(****************************************************************************************)
(* POU:		HLI3_HandlePlcSpindle                      									*)
(* Type:	Function Block																*)
(* Author: 	HR, MiB, TV																    *)
(* Date: 	10/11/10																	*)
(* Rev.: 	1.0																			*)
(* Rev.: 	1.6	14/10/23    															*)
(* ------------------------------------------------------------------------------------ *)
(* Desc:	Function block for handling technology functions of PLC spindles. It works	*)
(*			properly if there is a ation axis in the configuration. The logical 		*)
(*			axis no. 'n' of that axis is used to indetify that spindle in this function	*)
(*			block. This implies a spindle configuration like the folowing:				*)
(*				spdl_anzahl                         1	(maybe more?)					*)
(*				main_spindle_ax_nr                  n	(enter right value there)		*)
(*				main_spindle_name                   S									*)
(*				spindle_m_fct_free                  0									*)
(*				spindel[0].bezeichnung              S1									*)
(*				spindel[0].log_achs_nr              n	(enter right value there)		*)
(*				spindel[0].plc_control              1									*)
(*																						*)
(*			The function block may raise some errors specified by an error id:			*)
(*				+ 10000: axis number not valid!											*)
(*																						*)
(****************************************************************************************)
(* Date:	13/09/16																	*)
(* Author:	RCH																			*)
(* Rev:		1.1																			*)
(* ------------------------------------------------------------------------------------ *)
(* Desc 	Renamed, according to Tc2 version. This FB also works for CNC spindles with	*) 
(*			S or M functions set to inform PLC. 										*)
(****************************************************************************************)
(* Date:	13/09/16																	*)
(* Author:	RCH																			*)
(* Rev:		1.2																			*)
(* ------------------------------------------------------------------------------------ *)
(* Desc 	Introduced new input parameters 'bIsChannelSpecific' and 'nChannelNo' in 	*)
(*			order to make this FB work for PLC spindles which are sending synch.		*)
(*			requests via the channel specific section of the HLI. Here the spindle		*)
(* 			specific parameters have to be set as follows:								*)
(*				spindel[n].plc_control            1			(P-CHAN-00069)				*)
(*				spindel[n].log_achs_nr            m			(P-CHAN-00036)				*)
(*																						*)
(*			The logical axis number in P-CHAN-00036 used for such a spindle must not be	*)
(*			lower than one and must not be used by any other axis. This FB works if the	*)
(*			value of this logical axis number fits the parameter 'nHliAxisIdx' only!	*)
(* 																						*)
(*			In order to guarantee save HLI access the following new error codes have	*)
(*			been introduced:															*)
(*				+ 20000: Channel no lower than one!										*)
(*				+ 20001: Channel number exceeds number of configured channels.			*)
(*				+ 20002: No HLI data for channel.										*)
(****************************************************************************************)
(* Date:	14/01/22																	*)
(* Author:	TV																			*)
(* Rev:		1.3																			*)
(* ------------------------------------------------------------------------------------ *)
(* Desc:	bugfix in function to check nHLIAxisIdx and LogAxisId						*) 
(****************************************************************************************)
(* Date:	14/09/10																	*)
(* Author:	RCH																			*)
(* Rev:		1.4																			*)
(* ------------------------------------------------------------------------------------ *)
(* Desc 	Added optional handling of spindle gear change M functions M40 - M45.		*)
(****************************************************************************************)
(* Date:	14/09/12																	*)
(* Author:	RCH																			*)
(* Rev:		1.5																			*)
(* ------------------------------------------------------------------------------------ *)
(* Desc 	Fixed bug with spindle M functions send by the channel spec. section of the	*)
(*			HLI. So far the channel specific section was used for determining the value *)
(*			of  'nTechFctMaxidx'.														*)
(****************************************************************************************)
(* Date:	14/10/23																	*)
(* Author:	MiB																			*)
(* Rev:		1.6																			*)
(* ------------------------------------------------------------------------------------ *)
(* Desc 	Introduced parameter "nLogAxisNoChannelSpecific" which allows to use a plc  *)
(*			spindle without a simulation axis for the spindle. 				 			*)
(*			This paramater is only used if "bIsChannelSpecific == true"					*)
(*																						*)
(*				spindel[n].plc_control            1			(P-CHAN-00069)				*)
(*				spindel[n].log_achs_nr            m			(P-CHAN-00036)				*)
(*																						*)
(*			The logical axis number in P-CHAN-00036 used for such a spindle must not be	*)
(*			lower than one and must not be used by any other axis. This FB works if the	*)
(*			value of this logical axis number fits the parameter 						*)
(*			'nLogAxisNoChannelSpecific' only!											*)
(****************************************************************************************)
(* Date:	15/03/05																	*)
(* Author:	MiB																			*)
(* Rev:		1.7																			*)
(* ------------------------------------------------------------------------------------ *)
(* Desc 	Removed gearchange m functions from var_in_out							    *)
(*			Created new FB HLI3_SpindleTechnoGearchange									*)
(****************************************************************************************)
(*								Init Pointer to pM40..pM45								*)
(****************************************************************************************)
(* Date:	17/02/03																	*)
(* Author:	MiB																			*)
(* Rev:		1.7																			*)
(* ------------------------------------------------------------------------------------ *)
(* Desc 	Handling of late sync M functions. 											*)
(*			Usage of different structure TECHNO_UNIT_AX and TECHNO_UNIT_CH, depending 	*)
(*			on channel or axis specific specific interface 							 	*)
(****************************************************************************************)
(* Date:	19/04/19																	*)
(* Author:	TV																			*)
(* Rev:		1.8																			*)
(* ------------------------------------------------------------------------------------ *)
(* Desc 	Reset the M-Function flags after Reset										*)
(****************************************************************************************)


IF bFirstRun THEN
	bFirstRun := FALSE;
	pM40 := ADR(dummyM40);
	pM41 := ADR(dummyM41);
	pM42 := ADR(dummyM42);
	pM43 := ADR(dummyM43);
	pM44 := ADR(dummyM44);
	pM45 := ADR(dummyM45);	
END_IF

A_HandleTechno();

ACTION A_HandleTechno:

(****************************************************************************************)
(*								Cyclic reset of  error flag 							*)
(****************************************************************************************)
bError										:= FALSE;
nErrorId									:= 0;

(****************************************************************************************)
(*							  Check for valid logical axis no.							*)
(****************************************************************************************)
IF NOT bIsChannelSpecific AND NOT HLI3_CheckAxisValid(nHliAxisIdx := nHliAxisIdx) THEN
	bError									:= TRUE;
	nErrorId								:= 10000;
	RETURN;
END_IF

IF NOT HLI3_CheckChannelValid(nChannel := nHliChannelIdx) THEN
	bError									:= TRUE;
	nErrorId								:= 20000;
	RETURN;	
END_IF

(****************************************************************************************)
(*											Reset										*)
(****************************************************************************************)
fbRtrigChannelReset
	(CLK := bChannelReset);

IF fbRtrigChannelReset.Q THEN
	M_Reset(M03:=M03, M04:=M04,M05:=M05,M19:=M19);
END_IF

(****************************************************************************************)
(*									Receive requests from cnc							*)
(****************************************************************************************)
(* Look out for open technology function either on the channel or the axis specific		*)
(* section of the HLI, depending on parameter ''.										*)
IF bIsChannelSpecific THEN
	nOpenTechnoCount	:= gpCh[nHliChannelIdx]^.used_units_std_sync_r;
	nOpenTechnoCountLate:= gpCh[nHliChannelIdx]^.used_units_late_sync_r;
	
	nTechFctMaxidx 		:= gpCh[nHliChannelIdx]^.used_units_std_sync_r - 1;
	nTechFctMaxIdxLate 	:= gpCh[nHliChannelIdx]^.used_units_late_sync_r - 1;
ELSE
	nOpenTechnoCount	:= gpAx[nHliAxisIdx]^.used_units_std_sync_r;
	nOpenTechnoCountLate:= gpAx[nHliAxisIdx]^.used_units_late_sync_r;

	nTechFctMaxidx 		:= gpAx[nHliAxisIdx]^.used_units_std_sync_r - 1;
	nTechFctMaxIdxLate 	:= gpAx[nHliAxisIdx]^.used_units_late_sync_r - 1;		
END_IF

IF nOpenTechnoCount > 0 THEN
	FOR nLoop := 0 TO nTechFctMaxIdx DO
		(* Depending on the source determined by parameter 'bIsChannelSpecific', the		*)
		(* channel or axis specific section of the HLI will be examined.					*)
		IF bIsChannelSpecific THEN		
				
			M_HandleTechnoCh(ADR(gpCh[nHliChannelIdx]^.techno_unit_std_sync[nLoop]), M03 := M03, M04 := M04, M05 := M05, M19 := M19);												
		ELSE
			(* Get current axis specifc technology data *)			
			M_HandleTechnoAx(ADR(gpAx[nHliAxisIdx]^.techno_unit_std_sync[nLoop]), M03 := M03, M04 := M04, M05 := M05, M19 := M19);		
		END_IF																	
	END_FOR	
END_IF

IF nOpenTechnoCountLate > 0 THEN
	FOR nLoop := 0 TO nTechFctMaxIdxLate DO
		(* Depending on the source determined by parameter 'bIsChannelSpecific', the		*)
		(* channel or axis specific section of the HLI will be examined.					*)
		IF bIsChannelSpecific THEN			
			M_HandleTechnoCh(ADR(gpCh[nHliChannelIdx]^.techno_unit_late_sync[nLoop]), M03 := M03, M04 := M04, M05 := M05, M19 := M19);						
		ELSE
			(* Get current axis specifc technology data *)			
			M_HandleTechnoAx(ADR(gpAx[nHliAxisIdx]^.techno_unit_late_sync[nLoop]), M03 := M03, M04 := M04, M05 := M05, M19 := M19);	
		END_IF																	
	END_FOR	
END_IF

IF nOpenTechnoCountLate  = 0 AND nOpenTechnoCount = 0 THEN	
	M_Reset(M03:=M03, M04:=M04,M05:=M05,M19:=M19); 	 	
END_IF
END_ACTION

METHOD PROTECTED M_HandleTechnoAx
VAR_INPUT
	pActTechnoUnit:	POINTER TO TECHNO_UNIT_AX;	
END_VAR
VAR_IN_OUT
	/// Raises if the cnc program encounters a M03 for the relevant spindle. Reset this for acknowledge 
	M03: BOOL;
	/// Raises if the cnc program encounters a M04 for the relevant spindle. Reset this for acknowledge 
	M04: BOOL;
	/// Raises if the cnc program encounters a M05 for the relevant spindle. Reset this for acknowledge 
	M05: BOOL;
	/// Raises if the cnc program encounters a M19 for the relevant spindle. Reset this for acknowledge 
	M19: BOOL;
END_VAR
		
		(* Check request *)
		IF pActTechnoUnit^.please_rw AND
		   NOT pActTechnoUnit^.done_w
		THEN
			CASE UINT_TO_UDINT(pActTechnoUnit^.fkt_ctrl_r) OF
		     (* -------------------------------------------------------------------------- *)
			 (* Handle M function *)
			 HLI_INTF_M_FKT:
				pMProcess					:= ADR(pActTechnoUnit^.attribut_r.data[0]);
				
				IF (pMProcess > 0) AND bHandleGearChange THEN
					CASE pMProcess^.nr OF
					 40:	M_ManageAcknowledgement(ADR(M40_Internal), pM40, ADR(bAcknowledge));
					 41:	M_ManageAcknowledgement(ADR(M41_Internal), pM41, ADR(bAcknowledge));
					 42:	M_ManageAcknowledgement(ADR(M42_Internal), pM42, ADR(bAcknowledge));
					 43:	M_ManageAcknowledgement(ADR(M43_Internal), pM43, ADR(bAcknowledge));
					 44:	M_ManageAcknowledgement(ADR(M44_Internal), pM44, ADR(bAcknowledge));
					 45:	M_ManageAcknowledgement(ADR(M45_Internal), pM45, ADR(bAcknowledge));
					END_CASE
				END_IF
				
			 (* -------------------------------------------------------------------------- *)
			 (* Handle S function *)
			 HLI_INTF_SPINDEL:
				pSProcess					:= ADR(pActTechnoUnit^.attribut_r.data[0]);
				
				(* If we are working with spindle functions provided by the channel 		*)
				(* specific section of the HLI the logical axis number transmitted from the *)
				(* CNC must fit the one given in parameter 'nLogAxisNoChannelSpecific'!					*)												
				IF bIsChannelSpecific AND (UINT_TO_INT(pSProcess^.log_achs_nr) <> nLogAxisNoChannelSpecific) THEN
					RETURN;
				END_IF
	
				CASE pSProcess^.move_cmd OF
				 (* ----------------------------------------------------------------------- *)
				 0: (* M19 *)
					IF (pSProcess^.pos_cmd = 19) AND
					   NOT M19_Internal THEN
						nPosition			:= pSProcess^.pos;
						M19_Internal		:= TRUE;
						M19					:= TRUE;
					ELSE
						IF NOT M19 THEN
							M19_Internal	:= FALSE;
							bAcknowledge	:= TRUE;
						END_IF
					END_IF
	
				 (* ----------------------------------------------------------------------- *)
				 3: (* M03 *)
					nRevolution				:= pSProcess^.rev;
	
					IF NOT M03_Internal THEN
						M03_Internal		:= TRUE;
						M03					:= TRUE;
					ELSE
						IF NOT M03 THEN
							M03_Internal	:= FALSE;
							bAcknowledge	:= TRUE;
						END_IF
					END_IF
	
				 (* ----------------------------------------------------------------------- *)
				 4: (* M04 *)
					nRevolution				:= pSProcess^.rev;
	
					IF NOT M04_Internal THEN
						M04_Internal		:= TRUE;
						M04					:= TRUE;
					ELSE
						IF NOT M04 THEN
							M04_Internal	:= FALSE;
							bAcknowledge	:= TRUE;
						END_IF
					END_IF
	
				 (* ----------------------------------------------------------------------- *)
				 5: (* M05 *)
					IF NOT M05_Internal THEN
						M05_Internal		:= TRUE;
						M05					:= TRUE;
					ELSE
						IF NOT M05 THEN
							M05_Internal	:= FALSE;
							bAcknowledge	:= TRUE;
						END_IF
					END_IF
	
				END_CASE
			END_CASE
	
			(* Handle acknowledgement *)
			IF bAcknowledge THEN
				bAcknowledge				:= FALSE;
				nRevolution					:= 0;
				nPosition					:= 0;
				pActTechnoUnit^.please_rw 	:= FALSE;
		   		pActTechnoUnit^.done_w		:= TRUE;
			END_IF
		END_IF
END_METHOD

METHOD PROTECTED M_HandleTechnoCh
VAR_INPUT
	pActTechnoUnit:	POINTER TO TECHNO_UNIT_CH;
END_VAR
VAR_IN_OUT
	/// Raises if the cnc program encounters a M03 for the relevant spindle. Reset this for acknowledge 
	M03: BOOL;
	/// Raises if the cnc program encounters a M04 for the relevant spindle. Reset this for acknowledge 
	M04: BOOL;
	/// Raises if the cnc program encounters a M05 for the relevant spindle. Reset this for acknowledge 
	M05: BOOL;
	/// Raises if the cnc program encounters a M19 for the relevant spindle. Reset this for acknowledge 
	M19: BOOL;
END_VAR
		
		(* Check request *)
		IF pActTechnoUnit^.please_rw AND
		   NOT pActTechnoUnit^.done_w
		THEN
			CASE UINT_TO_UDINT(pActTechnoUnit^.fkt_ctrl_r) OF
		     (* -------------------------------------------------------------------------- *)
			 (* Handle M function *)
			 HLI_INTF_M_FKT:
				pMProcess					:= ADR(pActTechnoUnit^.attribut_r.data[0]);
				
				IF (pMProcess > 0) AND bHandleGearChange THEN
					CASE pMProcess^.nr OF
					 40:	M_ManageAcknowledgement(ADR(M40_Internal), pM40, ADR(bAcknowledge));
					 41:	M_ManageAcknowledgement(ADR(M41_Internal), pM41, ADR(bAcknowledge));
					 42:	M_ManageAcknowledgement(ADR(M42_Internal), pM42, ADR(bAcknowledge));
					 43:	M_ManageAcknowledgement(ADR(M43_Internal), pM43, ADR(bAcknowledge));
					 44:	M_ManageAcknowledgement(ADR(M44_Internal), pM44, ADR(bAcknowledge));
					 45:	M_ManageAcknowledgement(ADR(M45_Internal), pM45, ADR(bAcknowledge));
					END_CASE
				END_IF
				
			 (* -------------------------------------------------------------------------- *)
			 (* Handle S function *)
			 HLI_INTF_SPINDEL:
				pSProcess					:= ADR(pActTechnoUnit^.attribut_r.data[0]);
				
				(* If we are working with spindle functions provided by the channel 		*)
				(* specific section of the HLI the logical axis number transmitted from the *)
				(* CNC must fit the one given in parameter 'nLogAxisNoChannelSpecific'!					*)												
				IF bIsChannelSpecific AND (UINT_TO_INT(pSProcess^.log_achs_nr) <> nLogAxisNoChannelSpecific) THEN
					RETURN;
				END_IF
	
				CASE pSProcess^.move_cmd OF
				 (* ----------------------------------------------------------------------- *)
				 0: (* M19 *)
					IF (pSProcess^.pos_cmd = 19) AND
					   NOT M19_Internal THEN
						nPosition			:= pSProcess^.pos;
						M19_Internal		:= TRUE;
						M19					:= TRUE;
					ELSE
						IF NOT M19 THEN
							M19_Internal	:= FALSE;
							bAcknowledge	:= TRUE;
						END_IF
					END_IF
	
				 (* ----------------------------------------------------------------------- *)
				 3: (* M03 *)
					nRevolution				:= pSProcess^.rev;
	
					IF NOT M03_Internal THEN
						M03_Internal		:= TRUE;
						M03					:= TRUE;
					ELSE
						IF NOT M03 THEN
							M03_Internal	:= FALSE;
							bAcknowledge	:= TRUE;
						END_IF
					END_IF
	
				 (* ----------------------------------------------------------------------- *)
				 4: (* M04 *)
					nRevolution				:= pSProcess^.rev;
	
					IF NOT M04_Internal THEN
						M04_Internal		:= TRUE;
						M04					:= TRUE;
					ELSE
						IF NOT M04 THEN
							M04_Internal	:= FALSE;
							bAcknowledge	:= TRUE;
						END_IF
					END_IF
	
				 (* ----------------------------------------------------------------------- *)
				 5: (* M05 *)
					IF NOT M05_Internal THEN
						M05_Internal		:= TRUE;
						M05					:= TRUE;
					ELSE
						IF NOT M05 THEN
							M05_Internal	:= FALSE;
							bAcknowledge	:= TRUE;
						END_IF
					END_IF
	
				END_CASE
			END_CASE
	
			(* Handle acknowledgement *)
			IF bAcknowledge THEN
				bAcknowledge				:= FALSE;
				nRevolution					:= 0;
				nPosition					:= 0;
				pActTechnoUnit^.please_rw 	:= FALSE;
		   		pActTechnoUnit^.done_w		:= TRUE;
			END_IF
		END_IF
END_METHOD

{attribute 'object_name' := 'M_ManageAcknowledgement'}
METHOD PRIVATE M_ManageAcknowledgement
VAR_INPUT
	pInternal: POINTER TO BOOL;
	pPublic: POINTER TO BOOL;
	pAcknowledgement: POINTER TO BOOL;
END_VAR
IF NOT pInternal^ THEN
	pInternal^			:= TRUE;
	pPublic^			:= TRUE;	
ELSIF NOT pPublic^ THEN
	pInternal^			:= FALSE;
	pAcknowledgement^	:= TRUE;
END_IF
END_METHOD

METHOD M_Reset : BOOL
VAR_INPUT
END_VAR
VAR_IN_OUT	 
	M03: BOOL;	 
	M04: BOOL;	 
	M05: BOOL;	 
	M19: BOOL;
END_VAR
	nRevolution		:= 0;
	nPosition		:= 0;
	bAcknowledge	:= FALSE;
	M03				:= FALSE;
	M03_Internal	:= FALSE;
	M04				:= FALSE;
	M04_Internal	:= FALSE;
	M05				:= FALSE;
	M05_Internal	:= FALSE;
	M19				:= FALSE;
	M19_Internal	:= FALSE;	
	pM40^			:= FALSE;
	M40_Internal	:= FALSE;
	pM41^			:= FALSE;
	M41_Internal	:= FALSE;
	pM42^			:= FALSE;
	M42_Internal	:= FALSE;
	pM43^			:= FALSE;
	M43_Internal	:= FALSE;
	pM44^			:= FALSE;
	M44_Internal	:= FALSE;
	pM45^			:= FALSE;
	M45_Internal	:= FALSE;
END_METHOD

END_FUNCTION_BLOCK

// CNC/13 Spindle/HLI3_HandleSpindleTechnoGearchange
FUNCTION_BLOCK HLI3_HandleSpindleTechnoGearchange EXTENDS HLI3_HandleSpindleTechno
VAR_INPUT
END_VAR
VAR_OUTPUT
END_VAR
VAR_IN_OUT
		/// Raises if the cnc program encounters a M40 for the relevant spindle. Reset this for acknowledge 
	M40: BOOL;
	/// Raises if the cnc program encounters a M41 for the relevant spindle. Reset this for acknowledge 
	M41: BOOL;
	/// Raises if the cnc program encounters a M42 for the relevant spindle. Reset this for acknowledge 
	M42: BOOL;
	/// Raises if the cnc program encounters a M43 for the relevant spindle. Reset this for acknowledge 
	M43: BOOL;
	/// Raises if the cnc program encounters a M44 for the relevant spindle. Reset this for acknowledge 
	M44: BOOL;
	/// Raises if the cnc program encounters a M45 for the relevant spindle. Reset this for acknowledge 
	M45: BOOL;	
END_VAR
VAR
END_VAR

(* Date:	15/03/05																	*)
(* Author:	MiB																			*)
(* Rev:		1.0																			*)
(* ------------------------------------------------------------------------------------ *)
(* Desc 	Handling of spindle gear change M functions M40 - M45.						*)
(*			extends HLI3_SpindleTechno													*)
(*			overwrites the internal pointers to M40..M45 to VAR_IN_OUT					*)


SUPER^.pM40 := ADR(M40);
SUPER^.pM41 := ADR(M41);
SUPER^.pM42 := ADR(M42);
SUPER^.pM43 := ADR(M43);
SUPER^.pM44 := ADR(M44);
SUPER^.pM45 := ADR(M45);

A_HandleTechno();

END_FUNCTION_BLOCK

// CNC/13 Spindle/HLI3_MoveSpindle
///*********************************************************************************************************
///NAME.......................:	HLI3_MoveSpindle	
///DATUM....................:	24.5.2018
///AUTOR....................:	Michael Balsfulland (MiB) / TV
///VERSION................:	1.1
///				1.0 24.05.2018 Kopie von HLI_MoveSpindle
///				1.1 03.03.2019 Parametrierung der ControlUnit erst wenn command_semaphor_rw = false
 ///BESCHREIBUNG.:	 Spindel mit einer vorgegeben Geschwindigkeit starten oder Spindel stoppen
///......................: 	
///
///**********************************************************************************************************
 FUNCTION_BLOCK HLI3_MoveSpindle
VAR_INPUT
	/// HLI Index 
	nHliAxisIdx: INT;
	/// U/min 
	nSpeed: DINT;		// [u/min]
	/// steigende Flanke 
	bStart: BOOL;
	/// steigende Flanke 
	bStop: BOOL;
END_VAR
VAR_OUTPUT
	bBusy: BOOL;
	bError: BOOL;
	nErrID: INT;
	sErrText: STRING;
END_VAR
VAR
	pUnit: POINTER TO MC_CONTROL_EXT_TO_IPO;
	fbRTrigStart: R_TRIG;
	fbRTrigStop: R_TRIG;
	nState: INT;	 	
END_VAR

IF NOT (HLI3_CheckAxisValid(nHliAxisIdx := nHliAxisIdx)) THEN
		nState := -1;
		nErrID := 2;
		sErrText := 'Achsstruktur nicht vorhanden -> eventuell HLI Init nicht OK';
	RETURN;
END_IF

fbRTrigStart(clk := bStart);
IF fbRTrigStart.Q THEN
	bError := FALSE;
	nErrId := 0;
	sErrText := '';
	nState := 100;   (* Spindel starten *)
END_IF


fbRTrigStop(clk := bStop);
IF fbRTrigStop.Q THEN
	bError := FALSE;
	nErrId := 0;
	sErrText := '';
	nState := 200;  (* Spindel stoppen *)
END_IF

IF fbRTrigStop.Q OR fbRTrigStart.Q THEN   (* Grundzustände testen *)
	bBusy := TRUE;		
	IF gpAx[nHliAxisIdx]^.ipo_state.spindle_axis_r <> TRUE THEN
		nState := -1;
		nErrID := 3;
		sErrText := 'Achse ist kene Spindel';
	END_IF
END_IF

CASE nState OF


-1: (* Fehler *)
   	bError := TRUE;
	bBusy := FALSE;

0: (* IDLE *)
	bBusy := FALSE;


100: (* Spindel starten *)
	(* Check Override *)
	gpAx[nHliAxisIdx]^.ipo_mc_control.override.enable_w := TRUE;
	IF gpAx[nHliAxisIdx]^.ipo_mc_control.override.state_r = 0 THEN
		nState := -1;
		nErrID := 4;
		sErrText := 'Spindeloverride = 0';
	ELSE
		nState := 110;
	END_IF


110: (* Parametrieren des Aufrufs *)
	pUnit := ADR(gpAx[nHliAxisIdx]^.ipo_mc_control.ext_to_ipo);
	IF pUnit^.command_semaphor_rw = FALSE THEN
		IF (nSpeed > 0) THEN
			pUnit^.command_w.vb_prog   :=  nSpeed * 360 / 60 * 1000  ;(*Programmierter Satzvorschub in u/min*)
			pUnit^.command_w.dreh_info := 1;(* rechtslauf *)
		ELSE
			pUnit^.command_w.vb_prog   :=  -nSpeed * 360 / 60 * 1000  ;(*Programmierter Satzvorschub in u/min*)
			pUnit^.command_w.dreh_info := 0;(* linkslauf*)
		END_IF
		pUnit^.command_w.geo_gm_fkt    := 0;(*G- und M- Fkt.-Bitleiste*)
		pUnit^.command_w.satz_typ      := HLI_NC_MOVE_ENDLOS;(*Einer der Werte: HLI_NC_MOVE_LIN, HLI_NC_MOVREF, HLI_NC_MOVE_ENDLOS, HLI_NC_SPINDEL_STOP*)
		pUnit^.command_w.job_nr		   := 0;
		pUnit^.command_w.job_ackn      := FALSE;
	    pUnit^.command_semaphor_rw     := TRUE;
	    nState := 120;
	END_IF

	IF (nSpeed=0) THEN
		nState := -1;
		nErrID := 6;
		sErrText := 'Vorgabegeschwindigkeit = 0';
	END_IF

120: (* Start *)

	IF pUnit^.command_semaphor_rw = FALSE THEN
	    nState := 300;  (* checken Auftragsfehler *)
	END_IF



200: (* Spindel Stopp*)
	pUnit := ADR(gpAx[nHliAxisIdx]^.ipo_mc_control.ext_to_ipo);
	IF pUnit^.command_semaphor_rw = FALSE THEN
		pUnit^.command_w.satz_typ  := HLI_NC_SPINDEL_STOP;(*Einer der Werte: HLI_NC_MOVE_LIN, HLI_NC_MOVREF, HLI_NC_MOVE_ENDLOS, HLI_NC_SPINDEL_STOP*)		
		pUnit^.command_w.job_nr		   := 0;
		pUnit^.command_w.job_ackn      := FALSE;
		pUnit^.command_w.dreh_info := 0;(*Drehinformation*)
	   	pUnit^.command_semaphor_rw := TRUE;
	   	nState := 210;
	END_IF

210: (* Warten auf Stop *)
	IF pUnit^.command_semaphor_rw = FALSE THEN
	    nState := 300;   (* checken Auftragsfehler *)
	END_IF

300: (* checken Auftragsfehler *)
	IF (gpAx[nHliAxisIdx]^.ipo_state.spindle_order_error_r) THEN
		nState := -1;
		nErrID := 5;
		sErrText := 'Beauftragunsfehler Spindel';
	ELSE
		nState := 310;
	END_IF

310: (* Warten auf Solldrehzahl erreicht *)

	IF (gpAx[nHliAxisIdx]^.lr_state.rev_erreicht_r) THEN
		nState := 0;
	END_IF
END_CASE

END_FUNCTION_BLOCK

// CNC/Obsolete/HLI_MoveSpindle
///*********************************************************************************************************
///NAME.......................:	HLI_MoveSpindle	
///DATUM....................:	7.9.2009
///AUTOR....................:	Michael Balsfulland (MiB)
///VERSION................:	1.2
///				1.1 20.8.2010 MiB: kompletter Umbau auf Schrittkette mit Fehlerhandling
///				1.2 15.08.2017 MiB: BugFix: Linkslauf: Vorgabe der Drehzahl muss positiv erfolgen 
///BESCHREIBUNG.:	 Spindel mit einer vorgegeben Geschwindigkeit starten oder Spindel stoppen
///......................: 	
///
///**********************************************************************************************************
{attribute 'obsolete' := 'Please use HLI_MoveSpindle not valid!'}
FUNCTION_BLOCK HLI_MoveSpindle
VAR
	pUnit: POINTER TO MC_CONTROL_EXT_TO_IPO;
	fbRTrigStart: R_TRIG;
	fbRTrigStop: R_TRIG;
	nState: INT;
	/// Index of axis specific HLI area 
	nHliAxIfcIdx: UDINT;
END_VAR
VAR_INPUT
	/// Spindel Achssnummer 
	nLogAxisNr: UDINT;
	/// U/min 
	nSpeed: DINT;
	/// steigende Flanke 
	bStart: BOOL;
	/// steigende Flanke 
	bStop: BOOL;
END_VAR
VAR_OUTPUT
	bBusy: BOOL;
	bError: BOOL;
	nErrID: INT;
	sErrText: STRING;
END_VAR

fbRTrigStart(clk := bStart);
IF fbRTrigStart.Q THEN
	bError := FALSE;
	nErrId := 0;
	sErrText := '';
	nState := 100;   (* Spindel starten *)
END_IF


fbRTrigStop(clk := bStop);
IF fbRTrigStop.Q THEN
	bError := FALSE;
	nErrId := 0;
	sErrText := '';
	nState := 200;  (* Spindel stoppen *)
END_IF

nHliAxIfcIdx := nLogAxisNr - 1;

IF fbRTrigStop.Q OR fbRTrigStart.Q THEN   (* Grundzustände testen *)
	bBusy := TRUE;
	IF nLogAxisNr = 0 THEN
		nState := -1;
		nErrID := 1;
		sErrText := 'Spindel ID = 0';
	END_IF
	IF ADR(gpAx[nHliAxIfcIdx]^)  = 0  THEN
		nState := -1;
		nErrID := 2;
		sErrText := 'Achsstruktur nicht vorhanden -> eventuell HLI Init nicht OK';
	END_IF
	IF gpAx[nHliAxIfcIdx]^.ipo_state.spindle_axis_r <> TRUE THEN
		nState := -1;
		nErrID := 3;
		sErrText := 'Achse ist kene Spindel';
	END_IF
END_IF

CASE nState OF


-1: (* Fehler *)
   	bError := TRUE;
	bBusy := FALSE;

0: (* IDLE *)
	bBusy := FALSE;


100: (* Spindel starten *)
	(* Check Override *)
	gpAx[nHliAxIfcIdx]^.ipo_mc_control.override.enable_w := TRUE;
	IF gpAx[nHliAxIfcIdx]^.ipo_mc_control.override.state_r = 0 THEN
		nState := -1;
		nErrID := 4;
		sErrText := 'Spindeloverride = 0';
	ELSE
		nState := 110;
	END_IF


110: (* Parametrieren des Aufrufs *)
	pUnit := ADR(gpAx[nHliAxIfcIdx]^.ipo_mc_control.ext_to_ipo);
	IF (nSpeed > 0) THEN
		pUnit^.command_w.vb_prog   :=  nSpeed * 360 / 60 * 1000  ;(*Programmierter Satzvorschub in u/min*)
		pUnit^.command_w.dreh_info := 1;(* rechtslauf *)
	ELSE
		pUnit^.command_w.vb_prog   :=  -nSpeed * 360 / 60 * 1000  ;(*Programmierter Satzvorschub in u/min*)
		pUnit^.command_w.dreh_info := 0;(* linkslauf*)
	END_IF
	pUnit^.command_w.geo_gm_fkt    := 0;(*G- und M- Fkt.-Bitleiste*)
	pUnit^.command_w.satz_typ      := HLI_NC_MOVE_ENDLOS;(*Einer der Werte: HLI_NC_MOVE_LIN, HLI_NC_MOVREF, HLI_NC_MOVE_ENDLOS, HLI_NC_SPINDEL_STOP*)
	IF pUnit^.command_semaphor_rw = FALSE THEN
	    pUnit^.command_semaphor_rw := TRUE;
	    nState := 120;
	END_IF

	IF (nSpeed=0) THEN
		nState := -1;
		nErrID := 6;
		sErrText := 'Vorgabegeschwindigkeit = 0';
	END_IF

120: (* Start *)

	IF pUnit^.command_semaphor_rw = FALSE THEN
	    nState := 300;  (* checken Auftragsfehler *)
	END_IF



200: (* Spindel Stopp*)
	pUnit := ADR(gpAx[nHliAxIfcIdx]^.ipo_mc_control.ext_to_ipo);
	pUnit^.command_w.satz_typ  := HLI_NC_SPINDEL_STOP;(*Einer der Werte: HLI_NC_MOVE_LIN, HLI_NC_MOVREF, HLI_NC_MOVE_ENDLOS, HLI_NC_SPINDEL_STOP*)
	pUnit^.command_w.dreh_info := 0;(*Drehinformation*)
	IF pUnit^.command_semaphor_rw = FALSE THEN
	    pUnit^.command_semaphor_rw := TRUE;
	    nState := 210;
	END_IF

210: (* Warten auf Stop *)
	IF pUnit^.command_semaphor_rw = FALSE THEN
	    nState := 300;   (* checken Auftragsfehler *)
	END_IF

300: (* checken Auftragsfehler *)
	IF (gpAx[nHliAxIfcIdx]^.ipo_state.spindle_order_error_r) THEN
		nState := -1;
		nErrID := 5;
		sErrText := 'Beauftragunsfehler Spindel';
	ELSE
		nState := 310;
	END_IF

310: (* Warten auf Solldrehzahl erreicht *)

	IF (gpAx[nHliAxIfcIdx]^.lr_state.rev_erreicht_r) THEN
		nState := 0;
	END_IF


END_CASE


(*
IF nLogAxisNr <> 0 THEN
	IF pAC[nLogAxisNr] <> 0  THEN
		IF ADR(gpAx[nLogAxisNr]^) <> 0  THEN
			IF gpAx[nLogAxisNr]^.ipo_state.X_SpindleAxis = TRUE THEN

				(* command spindle revolution *)
				IF fbRTrigStart.Q THEN
					pCommand := ADR(gpAx[nLogAxisNr]^.ipo_mc_control.MCControlExtToIpo_ExtToIpo);
					IF (nSpeed > 0) THEN
						pCommand^.command_w.D_VbProg :=  DINT_TO_UDINT((nSpeed * 360 / 60) * 1000)  ;(*Programmierter Satzvorschub in u/min*)
  						pCommand^.command_w.W_DrehInfo := 1;(* rechtslauf *)
					ELSE
						pCommand^.command_w.D_VbProg :=  DINT_TO_UDINT((-nSpeed * 360 / 60) * 1000)  ;(*Programmierter Satzvorschub in u/min*)
						pCommand^.command_w.W_DrehInfo := 0;(* linkslauf*)
					END_IF
					pCommand^.command_w.D_GeoGmFkt := 0;(*G- und M- Fkt.-Bitleiste*)
					pCommand^.command_w.W_SatzTyp := HLI_NC_MOVE_ENDLOS;(*Einer der Werte: HLI_NC_MOVE_LIN, HLI_NC_MOVREF, HLI_NC_MOVE_ENDLOS, HLI_NC_SPINDEL_STOP*)
					pCommand^.command_semaphor_rw := TRUE;
				END_IF
				(* command spindle revolution *)
				IF fbRTrigStop.Q THEN
					pCommand := ADR(gpAx[nLogAxisNr]^.ipo_mc_control.MCControlExtToIpo_ExtToIpo);
					pCommand^.command_w.D_VbProg := 600000000;(*Programmierter Satzvorschub*)
					pCommand^.command_w.D_GeoGmFkt := 0;(*G- und M- Fkt.-Bitleiste*)

					pCommand^.command_w.W_SatzTyp := HLI_NC_SPINDEL_STOP;(*Einer der Werte: HLI_NC_MOVE_LIN, HLI_NC_MOVREF, HLI_NC_MOVE_ENDLOS, HLI_NC_SPINDEL_STOP*)
					pCommand^.command_w.W_DrehInfo := 0;(*Drehinformation*)
					pCommand^.command_semaphor_rw := TRUE;
				END_IF
			END_IF
		END_IF
	END_IF
END_IF
*)

END_FUNCTION_BLOCK

// CNC/13 Spindle/HLI3_ResetSpindle
FUNCTION HLI3_ResetSpindle : BOOL
VAR_INPUT
	/// axis number of spindle 
	nHliAxisIdx: INT;
END_VAR
VAR
	/// Index of axis specific HLI area 
	nHliAxIfcIdx: INT;
	SpdlState: BOOL;
	SpdlCommand: BOOL;
	ResetCmd: BOOL := FALSE;
	/// local pointer to data of actual axis 
	pResetUnit: POINTER TO MC_CONTROL_BOOL_UNIT;
END_VAR

HLI3_ResetSpindle := FALSE;

IF NOT HLI3_CheckAxisValid(nHliAxisIdx := nHliAxisIdx) THEN
	HLI3_ResetSpindle := FALSE;
	RETURN;
END_IF

	pResetUnit := ADR(gpAx[nHliAxisIdx]^.ipo_mc_control.spdl_reset);
	SpdlState  := pResetUnit^.state_r;

	IF ResetCmd = TRUE THEN
		pResetUnit^.command_w := TRUE;
		SpdlCommand           := pResetUnit^.command_w;
		HLI3_ResetSpindle          := SpdlState;
	END_IF

END_FUNCTION

// CNC/2 OperationMode/ModeManual/HLI3_LogicalAxisInManualMode
FUNCTION HLI3_LogicalAxisInManualMode : ARRAY[0..HLI_KEY_MAXIDX] OF UINT
VAR_INPUT
	nChan: INT;
END_VAR
VAR
	i: INT;
	n: INT;
END_VAR

(* 		  If no axis is in manual mode it returns 0           		*)
(* Author: MiB/TV                                         			*)
(*   Date: 16.07.2007                                         		*)
(*   Last: 05.04.2016                                        		*)
(*   Rev.: 1.1                                                 		*)
(* ================================================================= *)

IF (NOT HLI3_CheckChannelValid(nChannel := nChan)) THEN
	RETURN;
END_IF

n:= 0;
FOR i := 0 TO HLI_CH_AX_MAXIDX DO
  	IF (gpCh[nChan]^.bahn_state.coord_r[i].hb_display_r.state <> 0) THEN
		HLI3_LogicalAxisInManualMode[n] := gpCh[nChan]^.bahn_state.coord_r[i].log_achs_nr_r;
		IF n < HLI_KEY_MAXIDX THEN
			n := n+1;
		END_IF
	END_IF
END_FOR

END_FUNCTION

// CNC/2 OperationMode/ModeManual/HLI3_ManualActivation
FUNCTION_BLOCK HLI3_ManualActivation
VAR_INPUT
	bExecute: BOOL;
	/// Number of channel 
	nChan: INT;
	eManualType: E_CNC_ManualType;
	/// Increments -> 0 activates Tip mode 
	Inc: UDINT;
	/// Aufloesung des Achsverfahrwegs bei einer Handradumdrehung Einheit: 0.1um / Handradumdrehung
	nHBA_Res: DINT;
	Speed: UDINT;
	/// axis nr 
	nLogAxisNr: UINT;
	nInputParameterIdx: INT;
	nParameterRecordIdx : UINT;
END_VAR
VAR_OUTPUT
	bError: BOOL;
	bBusy: BOOL;
END_VAR
VAR_IN_OUT
	stManualModeControlElements: ST_ManualModeControlElements;
	stManualModeControlElementState: ST_ManualModeControlElementState;
END_VAR
VAR
	fbRtrigExec: R_TRIG;
	nState: INT;
	pActivation: POINTER TO MC_CONTROL_HB_ACTIVATION_UNIT;
	pJogParameter: POINTER TO MC_CONTROL_HB_JOG_PARAM_UNIT;
	pTipParameter: POINTER TO MC_CONTROL_HB_TIP_PARAM_UNIT;
	pHBHRParameter: POINTER TO MC_CONTROL_HB_HR_PARAM_UNIT;
	j: INT;
	bFreeControlElementFound: BOOL;
END_VAR

(* ========================================================= *)
(*    FUN: HLI_ManualActivation                       		 *)
(* --------------------------------------------------------- *)
(*   Desc:                                                   *)
(*   Author: CL TV MiB                                       *)
(*   Date: 18.11.2005                                        *)
(*   Last: 06.06.2017                                       *)
(*   Rev.: 6.2                                              *)
(* ========================================================= *)

IF NOT HLI3_CheckChannelValid(nChannel := nChan) OR nLogAxisNr = 0 THEN
	RETURN;
END_IF


fbRtrigExec(clk := bExecute);
IF fbRtrigExec.Q THEN
	bBusy := TRUE;
	bError := FALSE;
	nState := 10;
END_IF

CASE nState OF

	0: (* IDLE *)
		bBusy := FALSE;

	10:
		CASE eManualType OF
			E_CNC_ManualType.NoManualMode: 
				nState := 100;

			E_CNC_ManualType.Handwheel:
				nState := 30;

			E_CNC_ManualType.TippMode:
				nState := 40;

			E_CNC_ManualType.JogMode:
				nState := 50;

			E_CNC_ManualType.JoystickMode:
				nState := 40;

			E_CNC_ManualType.DigitalJoystick: 
				nState := 40;

		END_CASE

	30:(* Setze Handrad Parameter *)
		pHBHRParameter := ADR(gpCh[nChan]^.hb_mc_control.hr_parameter);
		IF NOT pHBHRParameter^.command_semaphor_rw THEN
			pHBHRParameter^.enable_w := TRUE;
			pHBHRParameter^.command_w.resolution  := nHBA_Res;
			pHBHRParameter^.command_w.log_achs_nr := nLogAxisNr;
			pHBHRParameter^.command_semaphor_rw := TRUE;
			nState := 100;
		END_IF

	40: (* Setze Parameter für den Tippbetrieb *)
		pTipParameter := ADR(gpCh[nChan]^.hb_mc_control.tip_parameter);
		IF NOT pTipParameter^.command_semaphor_rw THEN
			pTipParameter^.enable_w := TRUE;
			pTipParameter^.command_w.log_achs_nr := nLogAxisNr;
			pTipParameter^.command_w.speed       := Speed;			
			pTipParameter^.command_semaphor_rw := TRUE;
			nState := 100;
		END_IF

	50: (* Setze Parameter für den Jogbetrieb *)
		pJogParameter := ADR(gpCh[nChan]^.hb_mc_control.jog_parameter);
		IF NOT pJogParameter^.command_semaphor_rw THEN
			pJogParameter^.enable_w := TRUE;
			pJogParameter^.command_w.log_achs_nr := nLogAxisNr;
			pJogParameter^.command_w.distance    := Inc;
			pJogParameter^.command_w.speed       := Speed;
			pJogParameter^.command_semaphor_rw := TRUE;
			nState := 100;
		END_IF		
		
	100: 	(* Aktivierung der Bedienelementen für den Handbetrieb  *)
		pActivation := ADR(gpCh[nChan]^.hb_mc_control.activation);						
		IF 	NOT gpCh[nChan]^.hb_mc_control.activation.command_semaphor_rw AND 
			NOT gpCh[nChan]^.hb_mc_control.tip_parameter.command_semaphor_rw AND 
		   	NOT gpCh[nChan]^.hb_mc_control.jog_parameter.command_semaphor_rw AND 
		   	NOT gpCh[nChan]^.hb_mc_control.hr_parameter.command_semaphor_rw
		THEN 
			bFreeControlElementFound := FALSE;

			IF 	eManualType <> E_CNC_ManualType.Handwheel THEN 	
				FOR j := 0 TO HLI_KEY_MAXIDX DO
					IF stManualModeControlElementState.stKeyUnit[j].nLogAxisId = 0 THEN
							stManualModeControlElementState.stKeyUnit[j].nLogAxisId := nLogAxisNr;
							stManualModeControlElementState.stKeyUnit[j].nChan := nChan;
							stManualModeControlElementState.stKeyUnit[j].nInputParameterIdx := nInputParameterIdx;
							bFreeControlElementFound := TRUE;
						EXIT;
					END_IF 
				END_FOR
			ELSE
				FOR j := 0 TO HLI_HW_MAXIDX DO
					IF stManualModeControlElementState.stHWUnit[j].nLogAxisId = 0 THEN
							stManualModeControlElementState.stHWUnit[j].nLogAxisId := nLogAxisNr;
							stManualModeControlElementState.stHWUnit[j].nChan := nChan;
							stManualModeControlElementState.stHWUnit[j].nInputParameterIdx := nInputParameterIdx;
							bFreeControlElementFound := TRUE;
						EXIT;
					END_IF 
				END_FOR
			END_IF
							
			IF bFreeControlElementFound THEN
				pActivation^.enable_w := TRUE;
				pActivation^.command_w.log_achs_nr := nLogAxisNr;
				pActivation^.command_w.control_element := INT_TO_UINT(j+1);				
				pActivation^.command_w.parameter_index := nParameterRecordIdx;
		
				CASE eManualType OF
					E_CNC_ManualType.NoManualMode: 
						pActivation^.command_w.operation_mode := 0; 	(* 0 - No OP_Mode *)
		
					E_CNC_ManualType.Handwheel: 
						gpCh[0]^.hb_mc_control.handwheel_incs[j].command_w := stManualModeControlElements.nHandwheelInc[stManualModeControlElementState.stHWUnit[j].nInputParameterIdx];
						pActivation^.command_w.operation_mode := 1; 	(* 1 - Handwheel *)
		
					E_CNC_ManualType.TippMode: 
						pActivation^.command_w.operation_mode := 2; 	(* 2 - Tip Mode continous *)
		
					E_CNC_ManualType.JogMode: 
						pActivation^.command_w.operation_mode := 3; 	(* 3 - Jog Mode (incremental *)
		
					E_CNC_ManualType.JoystickMode: 
						pActivation^.command_w.operation_mode := 2; 	(* 2 - Tip Mode continous, auch für Analog Joystick *)
		
					E_CNC_ManualType.DigitalJoystick: 
						pActivation^.command_w.operation_mode := 2; 	(* 2 - Tip Mode continous, auch für Digital Joystick *)
		
				END_CASE
			
				pActivation^.command_semaphor_rw := TRUE;
				nState := 110;
			ELSE
				bError := TRUE;
				nState := 0;
			END_IF
		END_IF		

	110:	
		IF  NOT gpCh[nChan]^.hb_mc_control.activation.command_semaphor_rw  THEN 		
			nState := 0;
		END_IF
			
END_CASE

END_FUNCTION_BLOCK

// CNC/2 OperationMode/ModeManual/HLI3_ManualExecution
FUNCTION_BLOCK HLI3_ManualExecution
VAR_INPUT
	nChan: INT;
	/// number of the HB_KeyControlUnit 
	nKeyControlUnit: INT;
	/// static signal 
	bKeyPos: BOOL;
	/// static signal 
	bKeyNeg: BOOL;
END_VAR
VAR
	Cmd_Dir: E_HLI_MM_KEYDirection;
	Act_Dir: E_HLI_MM_KEYDirection;
END_VAR

(* ========================================================= *)
(*    FUN: HLI_ManualExecution                    		 		 *)
(* --------------------------------------------------------- *)
(*   Desc:                                                   *)
(*   Author: CL / TV                                         *)
(*   Date: 24.07.2015                                       *)
(*   Rev.: 6.0                                               *)
(* ========================================================= *)

(* flank detection second axis*)
gpCh[nChan]^.hb_mc_control.key[nKeyControlUnit].enable_w := TRUE;

IF (NOT bKeyPos AND NOT bKeyNeg) OR (bKeyPos AND Act_Dir = KEY_DIR_NEGATIVE) OR (bKeyNeg AND Act_Dir = KEY_DIR_POSITIVE) THEN
	Cmd_Dir := KEY_DIR_NOT_PRESSED;
	IF NOT gpCh[nChan]^.hb_mc_control.key[nKeyControlUnit].command_semaphor_rw AND Cmd_dir <> Act_Dir THEN
		gpCh[nChan]^.hb_mc_control.key[nKeyControlUnit].command_w.log_key_nr := DINT_TO_UINT(nKeyControlUnit)+1;
		gpCh[nChan]^.hb_mc_control.key[nKeyControlUnit].command_w.direction := KEY_DIR_NOT_PRESSED;
		gpCh[nChan]^.hb_mc_control.key[nKeyControlUnit].command_semaphor_rw := TRUE;
		Act_Dir := KEY_DIR_NOT_PRESSED;
	END_IF	
END_IF


IF bKeyPos AND Act_Dir = KEY_DIR_NOT_PRESSED THEN
	Cmd_Dir := KEY_DIR_POSITIVE;
	IF NOT gpCh[nChan]^.hb_mc_control.key[nKeyControlUnit].command_semaphor_rw AND Cmd_dir <> Act_Dir THEN
		gpCh[nChan]^.hb_mc_control.key[nKeyControlUnit].command_w.log_key_nr := DINT_TO_UINT(nKeyControlUnit)+1;
		gpCh[nChan]^.hb_mc_control.key[nKeyControlUnit].command_w.direction := KEY_DIR_POSITIVE;
		gpCh[nChan]^.hb_mc_control.key[nKeyControlUnit].command_semaphor_rw := TRUE;
		Act_Dir := KEY_DIR_POSITIVE;
	END_IF	
END_IF

IF bKeyNeg AND Act_Dir = KEY_DIR_NOT_PRESSED  THEN
	Cmd_Dir := KEY_DIR_NEGATIVE;
	IF NOT gpCh[nChan]^.hb_mc_control.key[nKeyControlUnit].command_semaphor_rw AND Cmd_dir <> Act_Dir THEN
		gpCh[nChan]^.hb_mc_control.key[nKeyControlUnit].command_w.log_key_nr := DINT_TO_UINT(nKeyControlUnit)+1;
		gpCh[nChan]^.hb_mc_control.key[nKeyControlUnit].command_w.direction := KEY_DIR_NEGATIVE;
		gpCh[nChan]^.hb_mc_control.key[nKeyControlUnit].command_semaphor_rw := TRUE;
		Act_Dir := KEY_DIR_NEGATIVE;
	END_IF	
END_IF

END_FUNCTION_BLOCK

// CNC/2 OperationMode/ModeManual/HLI3_ManualExecutionRapidMode
FUNCTION_BLOCK HLI3_ManualExecutionRapidMode
VAR_INPUT
	nChan: INT;
	/// number of the HB_KeyControlUnit 
	nKeyControlUnit: INT;
	/// static signal 
	bExecute: BOOL;
END_VAR
VAR
	pRapidKey: POINTER TO MC_CONTROL_HB_RAPID_KEY_UNIT;
	TONTimeOut: TON;
	fbRtrigExec: R_TRIG;
	fbFtrigExec: F_TRIG;
END_VAR

(* ========================================================= *)
(*    FUN: HLI_ManualExecution                               *)
(* --------------------------------------------------------- *)
(*   Desc:                                                   *)
(*   Author: TV                                              *)
(*   Date: 24.07.2015                                        *)
(*   Rev.: 6.0                                               *)
(* ========================================================= *)


IF nKeyControlUnit < 0 OR nKeyControlUnit > HLI_KEY_MAXIDX THEN
	RETURN;
END_IF;

pRapidKey := ADR(gpCh[nChan]^.hb_mc_control.rapid_key);
pRapidKey^.enable_w := TRUE;

IF NOT pRapidKey^.command_semaphor_rw THEN
	fbRtrigExec(clk := bExecute);
	fbFtrigExec(clk := bExecute);
END_IF

IF fbRtrigExec.Q THEN
	pRapidKey^.command_w.key_pressed := 1;
	pRapidKey^.command_w.log_key_nr := INT_TO_UINT(nKeyControlUnit)+1;
	pRapidKey^.command_semaphor_rw := TRUE;
END_IF


IF fbFtrigExec.Q THEN
	pRapidKey^.command_w.key_pressed := 0;
	pRapidKey^.command_w.log_key_nr := INT_TO_UINT(nKeyControlUnit)+1;
	pRapidKey^.command_semaphor_rw := TRUE;
END_IF

END_FUNCTION_BLOCK

// CNC/2 OperationMode/ModeManual/HLI3_ManualModeHandler
FUNCTION_BLOCK HLI3_ManualModeHandler
VAR_INPUT
	stManualModeParameter: ST_ManualModeParameter;
	stManualModeControlElements: ST_ManualModeControlElements;
	bReset: BOOL;
END_VAR
VAR_OUTPUT
	bInManualMode: BOOL;
	arrAxisInG201: ARRAY[0..HLI_KEY_MAXIDX] OF UINT;
	bBusy: BOOL;
	bError: BOOL;
	nErrorId: INT;
END_VAR
VAR_IN_OUT
	stManualModeControlElementState: ST_ManualModeControlElementState;
	stCmdModesStates: ST_CNCCmdModesStates;
END_VAR
VAR
	nState: INT;
	pString: POINTER TO STRING;
	pUnit: POINTER TO MC_CONTROL_MCM_MODE_STATE_UNIT;
	pCommand: POINTER TO HLI_PROC_TRANS_TO_MODE_STATE;
	pKey: POINTER TO MC_CONTROL_HB_KEY_UNIT;
	pIncr: POINTER TO MC_CONTROL_HB_TIP_PARAM_UNIT;
	stManualModeParameterOld: ST_ManualModeParameter;
	incOld: UINT;
	nManualTypOld: UINT;
	i: INT;
	bManual: BOOL;
	/// FBs for manual mode 
	ManualActivation: HLI3_ManualActivation;
	ManualExecution: ARRAY[0..HLI_KEY_MAXIDX] OF HLI3_ManualExecution;
	ManualExecutionRapidMode: ARRAY[0..HLI_KEY_MAXIDX] OF HLI3_ManualExecutionRapidMode;
	ActChannelModeOld: UDINT;
	TON_TimeOut: TON;
	nChan: INT;
	j: INT;
	bInJoystickMode: BOOL;
	nHliAxisIdx: INT;
	nControlUnit: INT;
	arrAxisInJoystickMode: ARRAY[0..HLI_KEY_MAXIDX] OF UINT;
	n: INT;
	bInit: BOOL;
	strInitParameter: STRING(HLI_IMCM_MODE_STATE_PARAM_STRL);
	strZeroOffset: STRING;
	fbRTrig: R_Trig;
	fbRTrigG200: R_Trig;
	fbRTrigG201: R_Trig;
	stManualOptionOld: ST_CNC_ManualOption;
	bClearState : BOOL;
END_VAR
VAR CONSTANT
	ErrID_1: INT := 1;
END_VAR

(* ========================================================= 	*)
(*     FB: HLI3_ManualModeHandler                           	*)
(* --------------------------------------------------------- 	*)
(*   Desc: Switch to Manual Mode and parametrize             	*)
(*   Author: MK / TV  /MiB                                      *)
(*   Date: 18.07.2002                                        	*)
(*   Last: 05.02.2021                                       	*)
(*   Rev.: 7.4	                                              	*)
(* ========================================================= 	*)
nChan := stManualModeParameter.stChannelParameter.nChanIdx;
IF (NOT HLI3_CheckChannelValid(nChannel := nChan) OR nChan = -1 )  THEN
	RETURN;
END_IF

IF 	CNCSystem.Channel[nChan].ActMode <> HLI_IMCM_MANUAL_MODE AND
	CNCSystem.Channel[nChan].ActMode <> HLI_IMCM_AUTOMATIC_MODE   AND
	CNCSystem.Channel[nChan].ActMode <> HLI_IMCM_MDI_MODE THEN
	//strInitParameterOld := '';	
	bManual := FALSE;
ELSE
	bManual := TRUE;
END_IF

bBusy := TRUE;

IF bReset THEN		
	bError := FALSE;
	nErrorID := 0;
	bInManualMode := FALSE;
END_IF

IF  ((NOT stCmdModesStates.stModes.Manual AND NOT gpCh[nChan]^.bahn_state.g201_active_r AND NOT gpCh[nChan]^.bahn_state.g200_active_r) OR 		
	CNCSystem.Channel[nChan].ActState = HLI_IMCM_PROCESS_ERROR) AND
	nState  <> 0 AND
	nState  <> 40 
	THEN 
		nState := 50; 
END_IF

Init();
G201();
Joystick();
CmdState();

fbRTrig(CLK:= stCmdModesStates.stModes.Manual); 
IF fbRTrig.Q THEN	
	strInitParameter:= '';
	nState 			:= 5;	
END_IF

fbRTrigG200(CLK:= gpCh[nChan]^.bahn_state.g200_active_r AND NOT gpCh[nChan]^.bahn_state.g201_active_r AND 
(gpCh[nCHan]^.channel_mc_control.mode_and_state.command_w.to_mode = HLI_IMCM_AUTOMATIC_MODE OR 
 gpCh[nCHan]^.channel_mc_control.mode_and_state.command_w.to_mode = HLI_IMCM_MDI_MODE OR 
 gpCh[nCHan]^.channel_mc_control.mode_and_state.command_w.to_mode = HLI_IMCM_REFERENCE_MODE));
IF fbRTrigG200.Q THEN	
	strInitParameter 	:= '';
	bClearState 		:= TRUE;
	nState 				:= 20;	
END_IF

fbRTrigG201(CLK:= gpCh[nChan]^.bahn_state.g201_active_r AND nstate = 0);   //nstate = 0 Modify 01.02.2021
IF fbRTrigG201.Q THEN	
	strInitParameter 	:= '';
	nState 				:= 20;	
END_IF

CASE nState OF
	0: (* IDLE *)
		bBusy 						:= FALSE;
		bInManualMode 				:= FALSE;
		bError 						:= FALSE;
		bClearState					:= FALSE;
		nErrorID 					:= 0;			
						
	 5: 	 	 
	 
	 	// 1. Zusatzstring zusammenbauen
			strInitParameter := '';	 					
		(* Activation of an manual mode string *)
		IF stManualModeParameter.stChannelParameter.stManualOption.bTrafoActive THEN
			strInitParameter := CONCAT(	strInitParameter,'$R$N#TRAFO ON$R$N');
		END_IF
			
		IF stManualModeParameter.stChannelParameter.stManualOption.bEcsActive THEN
			strInitParameter := CONCAT(strInitParameter,'$R$N#ECS ON$R$N');
		END_IF
			
		IF stManualModeParameter.stChannelParameter.stManualOption.bCAXActive THEN
			strInitParameter := CONCAT(strInitParameter,'$R$N#CAX$R$N');
		END_IF
						
		strInitParameter := CONCAT(stManualModeParameter.stChannelParameter.strInitParameter, strInitParameter);			
		strZeroOffset := '';
		CASE stManualModeParameter.stChannelParameter.stManualOption.eZeroOffset OF
			0: strZeroOffset := '$R$NG53';
			1: strZeroOffset := '$R$NG54';
			2: strZeroOffset := '$R$NG55';
			3: strZeroOffset := '$R$NG56';
			4: strZeroOffset := '$R$NG57';
			5: strZeroOffset := '$R$NG58';
			6: strZeroOffset := '$R$NG59';					
		ELSE				
			strZeroOffset  := CONCAT(strZeroOffset, '$R$NG159 = ');
			strZeroOffset  := CONCAT(strZeroOffset, INT_TO_STRING(stManualModeParameter.stChannelParameter.stManualOption.eZeroOffset));				
		END_CASE	
					
		strInitParameter := CONCAT(strInitParameter, strZeroOffset);	

		IF 	strInitParameter <> '' THEN				
			strInitParameter := CONCAT(strInitParameter,'$R$NG200');
		END_IF
																
		IF NOT gpCh[nCHan]^.channel_mc_control.mode_and_state.command_w.to_mode = HLI_IMCM_MANUAL_MODE THEN 
 			nState := 15;
	 	ELSIF strInitParameter <> ''  THEN
			nState := 10;
		END_IF
	
	10:											
		IF gpCh[nCHan]^.channel_mc_control.mode_and_state.command_semaphor_rw = FALSE THEN											
				gpCh[nCHan]^.channel_mc_control.mode_and_state.command_w.to_mode := HLI_IMCM_MANUAL_MODE ;
				gpCh[nCHan]^.channel_mc_control.mode_and_state.command_w.to_state := HLI_IMCM_PROCESS_SELECTED;
				gpCh[nCHan]^.channel_mc_control.mode_and_state.command_w.channel_number := INT_TO_UDINT(nChan+1);
				pString := ADR(gpCh[nCHan]^.channel_mc_control.mode_and_state.command_w.parameter);			
				pString^ := '';
				gpCh[nCHan]^.channel_mc_control.mode_and_state.command_semaphor_rw := TRUE;										
				nState := 15;
		END_IF		


15:		

	IF gpCh[nCHan]^.channel_mc_control.mode_and_state.command_semaphor_rw = FALSE THEN											
				gpCh[nCHan]^.channel_mc_control.mode_and_state.command_w.to_mode := HLI_IMCM_MANUAL_MODE ;
				gpCh[nCHan]^.channel_mc_control.mode_and_state.command_w.to_state := HLI_IMCM_PROCESS_ACTIVE;
				gpCh[nCHan]^.channel_mc_control.mode_and_state.command_w.channel_number := INT_TO_UDINT(nChan+1);
				pString := ADR(gpCh[nCHan]^.channel_mc_control.mode_and_state.command_w.parameter);			
				pString^ := strInitParameter;
				gpCh[nCHan]^.channel_mc_control.mode_and_state.command_semaphor_rw := TRUE;		
				
				n:= 0;					
								
				stManualOptionOld := stManualModeParameter.stChannelParameter.stManualOption;
				IF (CNCSystem.Channel[nChan].ActState = HLI_IMCM_PROCESS_ACTIVE OR gpCh[nChan]^.bahn_state.g201_active_r OR gpCh[nChan]^.bahn_state.g200_active_r) THEN
					nState := 20;
				END_IF
	END_IF	
			
	20: 	// Deactivation 											
				FOR j := 0 TO HLI_KEY_MAXIDX DO
					IF (stManualModeControlElementState.stKeyUnit[j].nChan = nChan) THEN
						stManualModeControlElementState.stKeyUnit[j].nChan := -1;
						stManualModeControlElementState.stKeyUnit[j].nLogAxisId := 0;
						stManualModeControlElementState.stKeyUnit[j].nInputParameterIdx := -1;
					END_IF													
				END_FOR
			
				FOR j := 0 TO HLI_HW_MAXIDX DO
					IF (stManualModeControlElementState.stHWUnit[j].nChan = nChan) THEN
						stManualModeControlElementState.stHWUnit[j].nChan := -1;
						stManualModeControlElementState.stHWUnit[j].nLogAxisId := 0;
						stManualModeControlElementState.stHWUnit[j].nInputParameterIdx := -1;
					END_IF													
				END_FOR	

		IF (n <= HLI_CH_AX_MAXIDX) THEN
			IF gpCh[nChan]^.bahn_state.coord_r[n].hb_display_r.control_element <> 0 THEN 
				IF NOT gpCh[nChan]^.hb_mc_control.activation.command_semaphor_rw THEN		
						gpCh[nChan]^.hb_mc_control.activation.command_w.log_achs_nr := gpCh[nChan]^.bahn_state.coord_r[n].log_achs_nr_r;
						gpCh[nChan]^.hb_mc_control.activation.command_w.control_element := 0;
						gpCh[nChan]^.hb_mc_control.activation.command_w.operation_mode := 0;
						
						IF (gpCh[nChan]^.bahn_state.coord_r[n].hb_display_r.operation_mode = 1) THEN
							stManualModeControlElementState.stHWUnit[gpCh[nChan]^.bahn_state.coord_r[n].hb_display_r.control_element-1].nChan := -1;
							stManualModeControlElementState.stHWUnit[gpCh[nChan]^.bahn_state.coord_r[n].hb_display_r.control_element-1].nLogAxisId :=0;
							stManualModeControlElementState.stHWUnit[gpCh[nChan]^.bahn_state.coord_r[n].hb_display_r.control_element-1].nInputParameterIdx := -1;	
						ELSE
							stManualModeControlElementState.stKeyUnit[gpCh[nChan]^.bahn_state.coord_r[n].hb_display_r.control_element-1].nChan := -1;
							stManualModeControlElementState.stKeyUnit[gpCh[nChan]^.bahn_state.coord_r[n].hb_display_r.control_element-1].nLogAxisId :=0;
							stManualModeControlElementState.stKeyUnit[gpCh[nChan]^.bahn_state.coord_r[n].hb_display_r.control_element-1].nInputParameterIdx := -1;						
						END_IF
						gpCh[nChan]^.hb_mc_control.activation.command_semaphor_rw := TRUE;
						nState := 21;					
				END_IF
			ELSE
				n := n + 1;
			END_IF				
		END_IF

		IF n >HLI_CH_AX_MAXIDX THEN
			nState := 28;
		END_IF
21: 
		IF 	NOT gpCh[nChan]^.hb_mc_control.activation.command_semaphor_rw THEN						
			n := n+1;
			nState := 20;
		END_IF
		
		IF n > HLI_CH_AX_MAXIDX THEN
			i		:= 0;			
			nState 	:= 28;
		END_IF																																		

28:		
		IF (gpCh[nCHan]^.channel_mc_control.mode_and_state.command_semaphor_rw = FALSE)  AND
			( CNCSystem.Channel[nChan].ActState = HLI_IMCM_PROCESS_ACTIVE OR gpCh[nChan]^.bahn_state.g201_active_r OR gpCh[nChan]^.bahn_state.g200_active_r) 
			THEN														
				ManualActivation(bExecute := FALSE, 
								stManualModeControlElements := stManualModeControlElements ,
								stManualModeControlElementState:= stManualModeControlElementState);
				i := 0;
				IF (gpCh[nChan]^.bahn_state.g200_active_r) THEN	
					nState := 30;
				END_IF						
		END_IF				
		
		IF bClearState THEN
		   nState := 0;
		END_IF
	
30: 	(* --- activate KeyControlUnits --- *)
		IF 	NOT stCmdModesStates.stModes.Manual AND 
			NOT gpCh[nChan]^.bahn_state.g201_active_r AND 
			NOT gpCh[nChan]^.bahn_state.g200_active_r 
			THEN 
			nState := 0;							
		ELSE							
			ManualActivation(bExecute := TRUE,
									nChan 			 := nChan,
									eManualType 	 := stManualModeParameter.stChannelParameter.eManualType,									
									stManualModeControlElementState:= stManualModeControlElementState,
									stManualModeControlElements := stManualModeControlElements,
									nInputParameterIdx := i,
									nParameterRecordIdx := stManualModeParameter.stAxisParameter.stControlUnit[i].nParameterRecordIdx,
									nHBA_Res 		 := stManualModeParameter.stChannelParameter.nHandwheelResolution,
									Inc 		     := stManualModeParameter.stChannelParameter.nInc,
									Speed 			 := stManualModeParameter.stAxisParameter.stControlUnit[i].nSpeed, // geändert alt nControlUnit
									nLogAxisNr 		 := stManualModeParameter.stAxisParameter.stControlUnit[i].nLogAxisNr); // geändert alt nControlUnit
			nState := 35;
		END_IF				
															
35: 	(* waiting for acknowledge *)
		ManualActivation(bExecute := FALSE, 
						stManualModeControlElements := stManualModeControlElements,
						stManualModeControlElementState:= stManualModeControlElementState);
		
		IF ManualActivation.bBusy = FALSE THEN
			IF ManualActivation.bError THEN
				nErrorId := ErrID_1;
				nState := 99;
			ELSE
				IF stManualModeParameter.stAxisParameter.stControlUnit[i+1].nLogAxisNr = 0 THEN
					i:=-1; (* reset the array counter *)

					stManualModeParameterOld    := stManualModeParameter;
					ActChannelModeOld   		:= cncsystem.Channel[nChan].ActMode;
				
					nState := 40;
				ELSE
					ManualActivation(bExecute := FALSE, 
									 stManualModeControlElements := stManualModeControlElements,
									 stManualModeControlElementState:= stManualModeControlElementState);
					nState := 30;
					i:= i+1;
				END_IF
			END_IF
		END_IF

40: 	(* endlich Handbetrieb *)
		bInManualMode := TRUE;
		
		IF (stManualModeParameter.stChannelParameter.eManualType <> E_CNC_ManualType.Handwheel) THEN
			FOR j := 0 TO HLI_KEY_MAXIDX DO
				IF stManualModeControlElementState.stKeyUnit[j].nChan = nChan AND stManualModeControlElementState.stKeyUnit[j].nLogAxisId <> 0 THEN				
					ManualExecution[j](	nChan := nChan,
									nKeyControlUnit := j,
									bKeyPos := stManualModeControlElements.stControlKeys[stManualModeControlElementState.stKeyUnit[j].nInputParameterIdx].bKeyPos,					// geändert 	nControlUnit
									bKeyNeg := stManualModeControlElements.stControlKeys[stManualModeControlElementState.stKeyUnit[j].nInputParameterIdx].bKeyNeg); (* no timeouts *)
									
					ManualExecutionRapidMode[j](nChan := nChan,
									nKeyControlUnit := j,
									bExecute := stManualModeControlElements.stControlKeys[stManualModeControlElementState.stKeyUnit[j].nInputParameterIdx].bKeyRapid); (* no timeouts *)
				END_IF
			END_FOR			
		ELSE				
			(* Handradincremente werden immer vom ersten Kanal entgegen genommen*)
			FOR j := 0 TO HLI_HW_MAXIDX DO
				IF (stManualModeControlElementState.stHWUnit[j].nChan = nChan AND stManualModeControlElementState.stHWUnit[j].nLogAxisId <>  0)  THEN 
					gpCh[0]^.hb_mc_control.handwheel_incs[j].command_w := stManualModeControlElements.nHandwheelInc[stManualModeControlElementState.stHWUnit[j].nInputParameterIdx];
				END_IF			
			END_FOR
		END_IF

		(* end of manual mode *)
		 IF (bManual = FALSE) OR           			                   
            NOT stCmdModesStates.stModes.Manual AND NOT gpCh[nChan]^.bahn_state.g201_active_r AND NOT gpCh[nChan]^.bahn_state.g200_active_r OR	                                                                                                                                                                                              
         	MEMCMP(ADR(stManualModeParameter),ADR(stManualModeParameterOld),SIZEOF(stManualModeParameter)-SIZEOF(stManualModeParameter.stChannelParameter.strInitParameter))<>0 OR
			MEMCMP(ADR(stManualOptionOld),ADR(stManualModeParameter.stChannelParameter.stManualOption),SIZEOF(stManualModeParameter.stChannelParameter.stManualOption))<>0 OR                                                      
            stManualModeParameter.stChannelParameter.strInitParameter <> stManualModeParameterOld.stChannelParameter.strInitParameter OR                                                          
            cncsystem.Channel[nChan].ActMode <> ActChannelModeOld OR                                       
            (CNCSystem.Channel[nChan].ActMode =  HLI_IMCM_MANUAL_MODE AND CNCSystem.Channel[nChan].ActState <> HLI_IMCM_PROCESS_ACTIVE) AND NOT gpCh[nChan]^.bahn_state.g201_active_r OR                                                   
            stManualModeParameter.stChannelParameter.eManualType = E_CNC_ManualType.NoManualMode
            THEN
		
				FOR j := 0 TO HLI_KEY_MAXIDX DO
					IF stManualModeControlElementState.stKeyUnit[j].nChan = nChan THEN
						ManualExecution[j](nChan := nChan,	nKeyControlUnit := j, bKeyPos := FALSE, bKeyNeg := FALSE); (* no timeouts *)		
					END_IF		
				END_FOR
						
				i:=1 (* resets the counter for the following deactivation *);			

				//stManualModeParameterOld 	:= stManualModeParameter;
	
				IF (bManual = FALSE) OR 
					//NOT gpCh[nChan]^.bahn_state.g200_active_r OR
					NOT gpCh[nChan]^.bahn_state.g201_active_r AND
					NOT gpCh[nChan]^.bahn_state.g200_active_r AND
					NOT stCmdModesStates.stModes.Manual OR
					stManualModeParameter.stChannelParameter.eManualType = E_CNC_ManualType.NoManualMode THEN 
					nState := 0;
				ELSIF (stManualModeParameter.stChannelParameter.strInitParameter <> stManualModeParameterOld.stChannelParameter.strInitParameter) OR 
					   (stManualOptionOld.bCAXActive <> stManualModeParameter.stChannelParameter.stManualOption.bCAXActive) OR
						(stManualOptionOld.bEcsActive <> stManualModeParameter.stChannelParameter.stManualOption.bEcsActive) OR
						(stManualOptionOld.bTrafoActive <> stManualModeParameter.stChannelParameter.stManualOption.bTrafoActive) OR
						(stManualOptionOld.bEcsActive <> stManualModeParameter.stChannelParameter.stManualOption.bEcsActive) OR
						(stManualOptionOld.eZeroOffset <> stManualModeParameter.stChannelParameter.stManualOption.eZeroOffset)
						 THEN								
					nState := 5;
				ELSIF gpCh[nChan]^.bahn_state.g200_active_r AND CNCSystem.Channel[nChan].ActMode = HLI_IMCM_AUTOMATIC_MODE THEN
					n	   := 0;	
					nState := 20;
				ELSE
					nState := 15;
				END_IF						
				
				bInManualMode := FALSE;				
		END_IF
		
		
50:		(* end of manual mode *)		
		FOR j := 0 TO HLI_KEY_MAXIDX DO
			IF stManualModeControlElementState.stKeyUnit[j].nChan = nChan THEN
				ManualExecution[j](nChan := nChan,	nKeyControlUnit := j, bKeyPos := FALSE, bKeyNeg := FALSE); (* no timeouts *)		
			END_IF		
		END_FOR
		nState := 0;				
				
99: 	(* error handling *)	
		bBusy := FALSE;
		bError := TRUE;
		
		(* end of manual mode *)
			IF NOT gpCh[nCHan]^.channel_mc_control.mode_and_state.command_semaphor_rw AND 
			CNCSystem.Channel[nChan].ActState <>  HLI_IMCM_PROCESS_ERROR
			THEN;
				gpCh[nCHan]^.channel_mc_control.mode_and_state.command_w.to_mode := HLI_IMCM_MANUAL_MODE ;
				gpCh[nCHan]^.channel_mc_control.mode_and_state.command_w.to_state := HLI_IMCM_PROCESS_SELECTED;
				gpCh[nCHan]^.channel_mc_control.mode_and_state.command_w.channel_number := INT_TO_UDINT(nChan+1);			
				gpCh[nCHan]^.channel_mc_control.mode_and_state.command_semaphor_rw := TRUE;	
			END_IF
			nState := 0;
		
		(* end of manual mode *)
		IF bManual = FALSE THEN
			bBusy := FALSE;
			nState := 0;
		END_IF

END_CASE

ACTION CmdState:
IF (NOT  gpCh[nCHan]^.channel_mc_control.mode_and_state.command_semaphor_rw) THEN    (* only if semaphor is FALSE...... *)
	IF stCmdModesStates.stStates.Selected THEN
		stCmdModesStates.stStates.Selected := FALSE;
		gpCh[nCHan]^.channel_mc_control.mode_and_state.command_w.to_mode := HLI_IMCM_MANUAL_MODE;
		gpCh[nCHan]^.channel_mc_control.mode_and_state.command_w.to_state := HLI_IMCM_PROCESS_SELECTED;		
		pString := ADR(gpCh[nCHan]^.channel_mc_control.mode_and_state.command_w.parameter);			
		pString^ := '';	
		gpCh[nCHan]^.channel_mc_control.mode_and_state.command_semaphor_rw := TRUE;
		nState := 0;		
	END_IF
	
	IF stCmdModesStates.stStates.Ready THEN
		stCmdModesStates.stStates.Ready := FALSE;
		gpCh[nCHan]^.channel_mc_control.mode_and_state.command_w.to_mode := HLI_IMCM_MANUAL_MODE;
		gpCh[nCHan]^.channel_mc_control.mode_and_state.command_w.to_state := HLI_IMCM_PROCESS_READY;		
		pString := ADR(gpCh[nCHan]^.channel_mc_control.mode_and_state.command_w.parameter);			
		pString^ := '';
		gpCh[nCHan]^.channel_mc_control.mode_and_state.command_semaphor_rw := TRUE;		
		nState := 0;
	END_IF
	
	IF stCmdModesStates.stStates.Active THEN
		stCmdModesStates.stStates.Active := FALSE;
		nState := 5;	
	END_IF
	
	IF stCmdModesStates.stStates.Hold THEN
		stCmdModesStates.stStates.Hold := FALSE;
		gpCh[nCHan]^.channel_mc_control.mode_and_state.command_w.to_mode := HLI_IMCM_MANUAL_MODE;
		gpCh[nCHan]^.channel_mc_control.mode_and_state.command_w.to_state := HLI_IMCM_PROCESS_HOLD;		
		gpCh[nCHan]^.channel_mc_control.mode_and_state.command_semaphor_rw := TRUE;
		nState := 0;		
	END_IF
	
	IF stCmdModesStates.stStates.Reset THEN
		stCmdModesStates.stStates.Reset := FALSE;
		gpCh[nCHan]^.channel_mc_control.mode_and_state.command_w.to_mode:= HLI_IMCM_MANUAL_MODE;
		gpCh[nCHan]^.channel_mc_control.mode_and_state.command_w.to_state := HLI_IMCM_PROCESS_RESETTING;		
		gpCh[nCHan]^.channel_mc_control.mode_and_state.command_semaphor_rw:= TRUE;
		nState := 0;		
	END_IF
END_IF
END_ACTION

ACTION G201:
(******** Parallelinterpolation mit G201 *************************************)
IF (CNCSystem.Channel[nChan].ActMode = HLI_IMCM_AUTOMATIC_MODE OR CNCSystem.Channel[nChan].ActMode = HLI_IMCM_MDI_MODE) 	
	AND (NOT stManualModeParameter.stChannelParameter.bG200ConfigurationViaPLC  OR gpCh[nChan]^.bahn_state.g201_active_r) THEN
	arrAxisInG201 := HLI3_LogicalAxisInManualMode(nCHan);
	FOR j := 0 TO HLI_KEY_MAXIDX DO
		stManualModeParameter.stAxisParameter.stControlUnit[j].nLogAxisNr := arrAxisInG201[j];
	END_FOR
ELSE
	FOR j := 0 TO HLI_KEY_MAXIDX DO
		arrAxisInG201[j] := 0;
	END_FOR
END_IF
END_ACTION

ACTION Init:
(* Clear all request from the HMI *)
IF gpCh[nChan]^.hb_mc_control.key[0].request_semaphor_rw THEN
	gpCh[nChan]^.hb_mc_control.key[0].request_semaphor_rw := FALSE;
END_IF

IF gpCh[nChan]^.hb_mc_control.activation.request_semaphor_rw THEN
	gpCh[nChan]^.hb_mc_control.activation.request_semaphor_rw := FALSE;
END_IF

IF gpCh[nChan]^.hb_mc_control.tip_parameter.request_semaphor_rw THEN
	gpCh[nChan]^.hb_mc_control.tip_parameter.request_semaphor_rw := FALSE;
END_IF

IF gpCh[nChan]^.hb_mc_control.jog_parameter.request_semaphor_rw THEN
	gpCh[nChan]^.hb_mc_control.jog_parameter.request_semaphor_rw := FALSE;
END_IF

IF NOT bInit THEN  
	gpCh[nChan]^.hb_mc_control.activation.enable_w := TRUE;
	FOR j := 0 TO HLI_HW_MAXIDX DO
		gpCh[nChan]^.hb_mc_control.handwheel_incs[j].enable_w  := TRUE;
	END_FOR
	bInit := TRUE;
END_IF
END_ACTION

ACTION Joystick:
IF stManualModeParameter.stChannelParameter.eManualType = E_CNC_ManualType.JoystickMode THEN

	bInJoystickMode := TRUE;	
	arrAxisInJoystickMode := HLI3_LogicalAxisInManualMode(nCHan);
		
	FOR j := 0 TO HLI_KEY_MAXIDX DO
		PRG_AnalogJoystick(	nLogAxisNr:= stManualModeParameter.stAxisParameter.stControlUnit[j].nLogAxisNr,
								Analog_Value:= stManualModeControlElements.stControlJoystickValue[j],
								AnalogValueMin:= stManualModeParameter.stJoystickParameter.AnalogValueMin,
								AnalogValueMax:= stManualModeParameter.stJoystickParameter.AnalogValueMax,
								AnalogValueZeroDeadBand:= stManualModeParameter.stJoystickParameter.AnalogValueZeroDeadBand,
								bKeyPos:= stManualModeControlElements.stControlKeys[j].bKeyPos,
								bKeyNeg:= stManualModeControlElements.stControlKeys[j].bKeyNeg);	
	END_FOR
																																					
ELSE
	(* Achsoverride wieder auf 100 % setzen *)
	IF bInJoystickMode THEN 
		nHliAxisIdx := -1;
		FOR j := 0 TO UINT_TO_INT(SIZEOF(arrAxisInJoystickMode)) DO
			FOR i := 0 TO UDINT_TO_INT(gNrAx-1) DO
				IF (gpAX[i]^.head.log_ax_nr_r = arrAxisInJoystickMode[j]) THEN
					nHliAxisIdx := i;	
					IF (nHliAxisIdx <> -1) THEN 
						HLI3_SetAxisOverride(nHliAxisIdx := nHliAxisIdx, nOverride := 1000);
						nHliAxisIdx := -1;
						arrAxisInJoystickMode[j] := 0;
					END_IF								
				END_IF
			END_FOR			
		END_FOR
		bInJoystickMode := FALSE;
	END_IF
END_IF
END_ACTION

END_FUNCTION_BLOCK

// CNC/2 OperationMode/ModeManual/PRG_AnalogJoystick
PROGRAM PRG_AnalogJoystick
VAR_INPUT
	nLogAxisNr: UINT;
	/// Actual Analog Value 
	Analog_Value: DINT;
	/// static signal : Analog Min Value 
	AnalogValueMin: DINT;
	/// static signal : Analog Max Value 
	AnalogValueMax: DINT;
	/// Dead Band for Zero Value 
	AnalogValueZeroDeadBand: DINT;
END_VAR
VAR_IN_OUT
	bKeyPos: BOOL;
	bKeyNeg: BOOL;
END_VAR
VAR
	/// Index of axis specific HLI area 
	nHliAxisIdx: INT;
	Norm_AnalogValue: LREAL;
	Zero_AnalogValue: LREAL;
	Override: LREAL;
END_VAR

(* ========================================================= *)
(*    Prog: Analog JoyStick			                  		 *)
(* --------------------------------------------------------- *)
(*   Desc:                                                   *)
(*   Author: TV	, MiB	                                         *)
(*   Date: 24.07.2015                                       *)
(*   Rev.: 6.0                                               *)
(* ========================================================= *)
	Norm_AnalogValue := (AnalogValueMax - AnalogValueMin);
	Zero_AnalogValue := AnalogValueMin + Norm_AnalogValue / 2;

	IF nLogAxisNr > 0 AND Norm_AnalogValue > 0 THEN
		nHliAxisIdx :=  HLI3_GetHliAxisIdx(UINT_TO_INT(nLogAxisNr));
		IF (nHliAxisIdx = -1) THEN
			RETURN;
		END_IF
		gpAx[nHliAxisIdx]^.ipo_mc_control.override.enable_w := TRUE;
		gpAx[nHliAxisIdx]^.ipo_mc_control.override_valid.enable_w := TRUE;
		gpAx[nHliAxisIdx]^.ipo_mc_control.override_valid.command_w := TRUE;
		Override := ABS(((Analog_Value  - AnalogValueMin) * 200 / Norm_AnalogValue)-100);

		IF Override > 100.0 THEN Override := 100.0; END_IF

		IF Analog_Value > Zero_AnalogValue THEN bKeyPos := TRUE; bKeyNeg := FALSE; ELSE bKeyPos := FALSE; END_IF
		IF Analog_Value < Zero_AnalogValue THEN bKeyNeg := TRUE; bKeyPos := FALSE; ELSE bKeyNeg := FALSE; END_IF

		IF Analog_Value > (Zero_AnalogValue - AnalogValueZeroDeadBand) AND Analog_Value < (Zero_AnalogValue + AnalogValueZeroDeadBand) THEN
			Override := 0;
			bKeyNeg := FALSE;
			bKeyPos := FALSE;
		END_IF

		gpAx[nHliAxisIdx]^.ipo_mc_control.override.command_w := LREAL_TO_UINT(Override * 10);
	END_IF

END_PROGRAM

// CNC/8 Mis/HLI3_GetHliAxisIdx
FUNCTION HLI3_GetHliAxisIdx : INT
VAR_INPUT
	nLogAxisId: INT;
END_VAR
VAR
	i: INT;
END_VAR

(* ========================================================= *)
(*    FUN: HLI3_GetHliAxisIdx                            *)
(* --------------------------------------------------------- *)
(*   Desc: returns teh HliAxisIdx for a given logical Axis id      	*)
(*   Author: MiB                                             *)
(*   Date: 5.8.2019                                        *)
(*   Rev.: 1.1                                               *)
(* ========================================================= *)
HLI3_GetHliAxisIdx := -1;
FOR i := 0 TO UDINT_TO_INT(gNrAx-1) DO
	IF nLogAxisId = UINT_TO_INT(gpAx[i]^.head.log_ax_nr_r) THEN
		HLI3_GetHliAxisIdx := i;
		RETURN;
	END_IF
END_FOR

END_FUNCTION

// CNC/3 Control/HLI3_SetAxisOverride
FUNCTION HLI3_SetAxisOverride : BOOL
VAR_INPUT
	/// number of Axis 
	nHliAxisIdx: INT;
	nOverride: UINT;
END_VAR

(* ========================================================= *)
(*    FUN: HLI_SetAxisOverride                               *)
(* --------------------------------------------------------- *)
(*   Desc: Set the Axis Override                             *)
(*   Author: TV                                              *)
(*   Date: 19.11.2018                                        *)
(*   Rev.: 1.2                                               *)
(*   Rev.: 1.1 MiB 19.11.2012 Tc3                            *)
(*   Rev.: 1.2 MiB 19.11.2018                                *)
(* ========================================================= *)
IF NOT (HLI3_CheckAxisValid(nHliAxisIdx := nHliAxisIdx)) THEN
	HLI3_SetAxisOverride := FALSE;
	RETURN;
END_IF


(* Limit the override *)
IF nOverride > 2000 THEN nOverride := 2000; END_IF  // TV 2018.11.19 valid maximum in cnc core is 2000
IF nOverride < 0 THEN nOverride := 0; END_IF

	gpAx[nHliAxisIdx]^.ipo_mc_control.override.enable_w  := TRUE;
	gpAx[nHliAxisIdx]^.ipo_mc_control.override.command_w := nOverride;

HLI3_SetAxisOverride := TRUE;

END_FUNCTION

// CNC/2 OperationMode/HLI3_AxisReset
FUNCTION HLI3_AxisReset : BOOL
VAR_INPUT
	/// Channel number 
	nChanNo: INT;
	/// Axis number 
	nHliAxisIdx: INT;
END_VAR
VAR
	/// local pointer to data of actual axis 
	pAxisData: POINTER TO HIGH_LEVEL_INTERFACE_AX;
END_VAR

(* ========================================================= *)
(*    FUN: HLI3_QuitAxisReset                                 *)
(* --------------------------------------------------------- *)
(*   Desc:                                                   *)
(* Author: MK , MiB                                          *)
(*   Date: 20.11.2012                                        *)
(*   Rev.: 1.1                                               *)
(* ========================================================= *)


HLI3_AxisReset := FALSE;
IF NOT HLI3_CheckAxisValid(nHliAxisIdx := nHliAxisIdx) THEN
	RETURN;
END_IF

IF gpAx[nHliAxisIdx] = 0 THEN
	RETURN;
END_IF


(* get pointer to axis data *)
pAxisData := gpAx[nHliAxisIdx];
IF pAxisData^.ipo_state.cnc_channel_r = INT_TO_UINT(nChanNo) THEN (* it's an axis of the channel *)
	(* is a reset commanded *)
	IF pAxisData^.ipo_lc_control.plc_reset.command_r = TRUE THEN
		(* quit this reset *)
		pAxisData^.ipo_lc_control.plc_reset.state_w := TRUE;	
		HLI3_AxisReset := TRUE;
	END_IF
END_IF

END_FUNCTION

// CNC/2 OperationMode/HLI3_ChannelModeAuto
FUNCTION HLI3_ChannelModeAuto : BOOL
VAR_INPUT	
	nChanIdx: INT;
	ProgramName: STRING(HLI_IMCM_MODE_STATE_PARAM_STRL);			
END_VAR
VAR_IN_OUT
	stCmdModesStates    : ST_CNCCmdModesStates;	
END_VAR
VAR
	pString: POINTER TO STRING(HLI_IMCM_MODE_STATE_PARAM_STRL);
END_VAR

(* ========================================================= *)
(*    FUN: HLI_ChannelModeAuto                               *)
(* --------------------------------------------------------- *)
(*   Desc: switch channel to Automatic mode / xxx            *)
(*   Author: MK,MiB, TV                                      *)
(*   Date: 03.03.2017                                        *)
(*   Rev.: 1.5                                               *)
(* ========================================================= *)

IF (NOT gpCh[nChanIdx]^.channel_mc_control.mode_and_state.command_semaphor_rw) THEN    (* only if semaphor is FALSE...... *)
	IF stCmdModesStates.stStates.Selected THEN
		stCmdModesStates.stStates.Selected := FALSE;
		gpCh[nChanIdx]^.channel_mc_control.mode_and_state.command_w.to_mode := HLI_IMCM_AUTOMATIC_MODE;
		gpCh[nChanIdx]^.channel_mc_control.mode_and_state.command_w.to_state := HLI_IMCM_PROCESS_SELECTED;	
		pString := ADR(gpCh[nChanIdx]^.channel_mc_control.mode_and_state.command_w.parameter);			
		pString^ := ProgramName;				
		gpCh[nChanIdx]^.channel_mc_control.mode_and_state.command_semaphor_rw  := TRUE;		
	END_IF
	
	IF stCmdModesStates.stStates.Ready THEN
		stCmdModesStates.stStates.Ready := FALSE;
		gpCh[nChanIdx]^.channel_mc_control.mode_and_state.command_w.to_mode := HLI_IMCM_AUTOMATIC_MODE;
		gpCh[nChanIdx]^.channel_mc_control.mode_and_state.command_w.to_state := HLI_IMCM_PROCESS_READY;		
		pString := ADR(gpCh[nChanIdx]^.channel_mc_control.mode_and_state.command_w.parameter);			
		pString^ := ProgramName;				
		gpCh[nChanIdx]^.channel_mc_control.mode_and_state.command_semaphor_rw  := TRUE;		
	END_IF
	
	IF stCmdModesStates.stStates.Active THEN
		stCmdModesStates.stStates.Active := FALSE;
		gpCh[nChanIdx]^.channel_mc_control.mode_and_state.command_w.to_mode := HLI_IMCM_AUTOMATIC_MODE;
		gpCh[nChanIdx]^.channel_mc_control.mode_and_state.command_w.to_state := HLI_IMCM_PROCESS_ACTIVE;		
		pString := ADR(gpCh[nChanIdx]^.channel_mc_control.mode_and_state.command_w.parameter);			
		pString^ := ProgramName;				
		gpCh[nChanIdx]^.channel_mc_control.mode_and_state.command_semaphor_rw  := TRUE;		
	END_IF
	
	IF stCmdModesStates.stStates.Hold THEN
		stCmdModesStates.stStates.Hold:= FALSE;
		gpCh[nChanIdx]^.channel_mc_control.mode_and_state.command_w.to_mode:= HLI_IMCM_AUTOMATIC_MODE;
		gpCh[nChanIdx]^.channel_mc_control.mode_and_state.command_w.to_state := HLI_IMCM_PROCESS_HOLD;		
		gpCh[nChanIdx]^.channel_mc_control.mode_and_state.command_semaphor_rw  := TRUE;
	END_IF
	
	IF stCmdModesStates.stStates.Reset THEN
		stCmdModesStates.stStates.Reset := FALSE;
		gpCh[nChanIdx]^.channel_mc_control.mode_and_state.command_w.to_mode := HLI_IMCM_AUTOMATIC_MODE;
		gpCh[nChanIdx]^.channel_mc_control.mode_and_state.command_w.to_state:= HLI_IMCM_PROCESS_RESETTING;		
		gpCh[nChanIdx]^.channel_mc_control.mode_and_state.command_semaphor_rw  := TRUE;		
	END_IF
	
	HLI3_ChannelModeAuto := TRUE;
ELSE
	HLI3_ChannelModeAuto := FALSE;
END_IF

END_FUNCTION

// CNC/2 OperationMode/HLI3_ChannelModeManual
FUNCTION HLI3_ChannelModeManual : BOOL
VAR_INPUT	
	nChanIdx: INT;	
END_VAR

VAR_IN_OUT
	stCmdModesStates    : ST_CNCCmdModesStates;	
END_VAR

VAR
	pString: POINTER TO STRING;
END_VAR

(* ========================================================= *)
(*    FUN: HLI_ChannelModeManual                             *)
(* --------------------------------------------------------- *)
(*   Desc: switch channel to Manual mode / xxx               *)
(*   Author: MK, MiB, TV, RCH                                *)
(*   Date: 03.03.2017                                        *)
(*   Rev.: 1.5                                               *)
(* ========================================================= *)

IF (NOT  gpCh[nChanIdx]^.channel_mc_control.mode_and_state.command_semaphor_rw) THEN    (* only if semaphor is FALSE...... *)
	IF stCmdModesStates.stStates.Selected THEN
		stCmdModesStates.stStates.Selected := FALSE;
		gpCh[nChanIdx]^.channel_mc_control.mode_and_state.command_w.to_mode := HLI_IMCM_MANUAL_MODE;
		gpCh[nChanIdx]^.channel_mc_control.mode_and_state.command_w.to_state := HLI_IMCM_PROCESS_SELECTED;		
		pString := ADR(gpCh[nChanIdx]^.channel_mc_control.mode_and_state.command_w.parameter);			
		pString^ := '';	
		gpCh[nChanIdx]^.channel_mc_control.mode_and_state.command_semaphor_rw := TRUE;		
	END_IF
	
	IF stCmdModesStates.stStates.Ready THEN
		stCmdModesStates.stStates.Ready := FALSE;
		gpCh[nChanIdx]^.channel_mc_control.mode_and_state.command_w.to_mode := HLI_IMCM_MANUAL_MODE;
		gpCh[nChanIdx]^.channel_mc_control.mode_and_state.command_w.to_state := HLI_IMCM_PROCESS_READY;		
		pString := ADR(gpCh[nChanIdx]^.channel_mc_control.mode_and_state.command_w.parameter);			
		pString^ := '';
		gpCh[nChanIdx]^.channel_mc_control.mode_and_state.command_semaphor_rw := TRUE;		
	END_IF
	
	IF stCmdModesStates.stStates.Active THEN
		stCmdModesStates.stStates.Active := FALSE;
		gpCh[nChanIdx]^.channel_mc_control.mode_and_state.command_w.to_mode := HLI_IMCM_MANUAL_MODE;
		gpCh[nChanIdx]^.channel_mc_control.mode_and_state.command_w.to_state := HLI_IMCM_PROCESS_ACTIVE;		
		pString := ADR(gpCh[nChanIdx]^.channel_mc_control.mode_and_state.command_w.parameter);			
		pString^ := '';						
		gpCh[nChanIdx]^.channel_mc_control.mode_and_state.command_semaphor_rw := TRUE;	
	END_IF
	
	IF stCmdModesStates.stStates.Hold THEN
		stCmdModesStates.stStates.Hold := FALSE;
		gpCh[nChanIdx]^.channel_mc_control.mode_and_state.command_w.to_mode := HLI_IMCM_MANUAL_MODE;
		gpCh[nChanIdx]^.channel_mc_control.mode_and_state.command_w.to_state := HLI_IMCM_PROCESS_HOLD;		
		gpCh[nChanIdx]^.channel_mc_control.mode_and_state.command_semaphor_rw := TRUE;		
	END_IF
	
	IF stCmdModesStates.stStates.Reset THEN
		stCmdModesStates.stStates.Reset := FALSE;
		gpCh[nChanIdx]^.channel_mc_control.mode_and_state.command_w.to_mode:= HLI_IMCM_MANUAL_MODE;
		gpCh[nChanIdx]^.channel_mc_control.mode_and_state.command_w.to_state := HLI_IMCM_PROCESS_RESETTING;		
		gpCh[nChanIdx]^.channel_mc_control.mode_and_state.command_semaphor_rw:= TRUE;		
	END_IF

	HLI3_ChannelModeManual := TRUE;
ELSE
	HLI3_ChannelModeManual := FALSE;
END_IF

END_FUNCTION

// CNC/2 OperationMode/HLI3_ChannelModeMDI
FUNCTION HLI3_ChannelModeMDI : BOOL
VAR_INPUT	
	nChanIdx: INT;	
	/// pointer to the MDI program string 
	pMDIString: POINTER TO STRING(HLI_IMCM_MODE_STATE_PARAM_STRL);
END_VAR

VAR_IN_OUT
	stCmdModesStates    : ST_CNCCmdModesStates;	
END_VAR
VAR
	pString: POINTER TO STRING(HLI_IMCM_MODE_STATE_PARAM_STRL);
END_VAR

(* ========================================================= *)
(*    FUN: HLI_ChannelModeMDI                                *)
(* --------------------------------------------------------- *)
(*   Desc: switch channel to MDI mode / xxx                  *)
(*   Author: MK, TV, MiB, Rch                                *)
(*   Date: 18.07.2002                                        *)
(*   Last: 03.03.2017                      				     *)
(*   Rev.: 1.7                                               *)
(* ========================================================= *)

IF (NOT gpCh[nChanIdx]^.channel_mc_control.mode_and_state.command_semaphor_rw) THEN  (* only if semaphor is FALSE...... *)

	IF stCmdModesStates.stStates.Selected THEN
		stCmdModesStates.stStates.Selected := FALSE;
		gpCh[nChanIdx]^.channel_mc_control.mode_and_state.command_w.to_mode := HLI_IMCM_MDI_MODE;
		gpCh[nChanIdx]^.channel_mc_control.mode_and_state.command_w.to_state := HLI_IMCM_PROCESS_SELECTED;
		pString := ADR(gpCh[nChanIdx]^.channel_mc_control.mode_and_state.command_w.parameter);					
		pString^ := pMDIString^;
		gpCh[nChanIdx]^.channel_mc_control.mode_and_state.command_semaphor_rw := TRUE;		
	END_IF
	
	IF stCmdModesStates.stStates.Ready THEN
		stCmdModesStates.stStates.Ready := FALSE;
		gpCh[nChanIdx]^.channel_mc_control.mode_and_state.command_w.to_mode:= HLI_IMCM_MDI_MODE;
		gpCh[nChanIdx]^.channel_mc_control.mode_and_state.command_w.to_state := HLI_IMCM_PROCESS_READY;		
		gpCh[nChanIdx]^.channel_mc_control.mode_and_state.command_semaphor_rw := TRUE;		
	END_IF
	
	IF stCmdModesStates.stStates.Active THEN
		stCmdModesStates.stStates.Active := FALSE;
		gpCh[nChanIdx]^.channel_mc_control.mode_and_state.command_w.to_mode := HLI_IMCM_MDI_MODE;
		gpCh[nChanIdx]^.channel_mc_control.mode_and_state.command_w.to_state := HLI_IMCM_PROCESS_ACTIVE;
		pString := ADR(gpCh[nChanIdx]^.channel_mc_control.mode_and_state.command_w.parameter);					
		pString^ := pMDIString^;
		gpCh[nChanIdx]^.channel_mc_control.mode_and_state.command_semaphor_rw := TRUE;		
	END_IF
	
	IF stCmdModesStates.stStates.Hold THEN
		stCmdModesStates.stStates.Hold := FALSE;
		gpCh[nChanIdx]^.channel_mc_control.mode_and_state.command_w.to_mode := HLI_IMCM_MDI_MODE;
		gpCh[nChanIdx]^.channel_mc_control.mode_and_state.command_w.to_state:= HLI_IMCM_PROCESS_HOLD;		
		gpCh[nChanIdx]^.channel_mc_control.mode_and_state.command_semaphor_rw := TRUE;		
	END_IF
	
	IF stCmdModesStates.stStates.Reset THEN
		stCmdModesStates.stStates.Reset := FALSE;
		gpCh[nChanIdx]^.channel_mc_control.mode_and_state.command_w.to_mode := HLI_IMCM_MDI_MODE;
		gpCh[nChanIdx]^.channel_mc_control.mode_and_state.command_w.to_state := HLI_IMCM_PROCESS_RESETTING;		
		gpCh[nChanIdx]^.channel_mc_control.mode_and_state.command_semaphor_rw := TRUE;		
	END_IF
	HLI3_ChannelModeMDI := TRUE;	
ELSE
	HLI3_ChannelModeMDI := FALSE;
END_IF

END_FUNCTION

// CNC/2 OperationMode/HLI3_ChannelModeReference
FUNCTION HLI3_ChannelModeReference : BOOL
VAR_INPUT	
	nChanIdx: INT;	
	/// the referencing string 
	sRefPosString: STRING(HLI_IMCM_MODE_STATE_PARAM_STRL);	
END_VAR

VAR_IN_OUT
	stCmdModesStates    : ST_CNCCmdModesStates;	
END_VAR

VAR
	pString: POINTER TO STRING(HLI_IMCM_MODE_STATE_PARAM_STRL);
END_VAR

(* ========================================================= *)
(*    FUN: HLI_ChannelModeReference                          *)
(* --------------------------------------------------------- *)
(*   Desc: switch channel to Reference mode / xxx            *)
(*   Author: MK, MiB, TV                                     *)
(*   Date: 03.03.2017                                        *)
(*   Rev.: 1.5                                               *)
(* ========================================================= *)


(************************************************************
	RefPosString:
	Element: parameter ( ASCII char set, Länge:256 Zeichen)

	Vorgabe zur Parametrierung der Referenzpunktfahrt.

	Ist dieser STRING leer, so wird defaultmäßig das
	Automatikprogramm "rpf.nc" angewählt.

	Ansonsten kann durch explizite Angabe der Achsen und
	Zeitpunkt im Format "G74
	<Achsbezeichner_1><Zeitpunkt_1> ...
	<Achsbezeichner_n><Zeitpunkt_n>"
	eine individuelle Referenzpunktfahrt vorgegeben werden.
*************************************************************)

IF (NOT gpCh[nChanIdx]^.channel_mc_control.mode_and_state.command_semaphor_rw) THEN  (* only if semaphor is FALSE...... *)
	IF stCmdModesStates.stStates.Selected THEN
		stCmdModesStates.stStates.Selected := FALSE;
		gpCh[nChanIdx]^.channel_mc_control.mode_and_state.command_w.to_mode := HLI_IMCM_REFERENCE_MODE;
		gpCh[nChanIdx]^.channel_mc_control.mode_and_state.command_w.to_state := HLI_IMCM_PROCESS_SELECTED;		
		gpCh[nChanIdx]^.channel_mc_control.mode_and_state.command_semaphor_rw := TRUE;	
	END_IF
	
	IF stCmdModesStates.stStates.Ready THEN
		stCmdModesStates.stStates.Ready := FALSE;
		gpCh[nChanIdx]^.channel_mc_control.mode_and_state.command_w.to_mode := HLI_IMCM_REFERENCE_MODE;
		gpCh[nChanIdx]^.channel_mc_control.mode_and_state.command_w.to_state := HLI_IMCM_PROCESS_READY;		
		pString := ADR(gpCh[nChanIdx]^.channel_mc_control.mode_and_state.command_w.parameter);	
		gpCh[nChanIdx]^.channel_mc_control.mode_and_state.command_semaphor_rw := TRUE;		
	END_IF
	
	IF stCmdModesStates.stStates.Active THEN
		stCmdModesStates.stStates.Active := FALSE;
		gpCh[nChanIdx]^.channel_mc_control.mode_and_state.command_w.to_mode := HLI_IMCM_REFERENCE_MODE;
		gpCh[nChanIdx]^.channel_mc_control.mode_and_state.command_w.to_state := HLI_IMCM_PROCESS_ACTIVE;		
		pString := ADR(gpCh[nChanIdx]^.channel_mc_control.mode_and_state.command_w.parameter);	
		pString^ := sRefPosString;
		gpCh[nChanIdx]^.channel_mc_control.mode_and_state.command_semaphor_rw:= TRUE;		
	END_IF
	
	IF stCmdModesStates.stStates.Hold THEN
		stCmdModesStates.stStates.Hold := FALSE;
		gpCh[nChanIdx]^.channel_mc_control.mode_and_state.command_w.to_mode := HLI_IMCM_REFERENCE_MODE;
		gpCh[nChanIdx]^.channel_mc_control.mode_and_state.command_w.to_state := HLI_IMCM_PROCESS_HOLD;		
		gpCh[nChanIdx]^.channel_mc_control.mode_and_state.command_semaphor_rw := TRUE;		
	END_IF
	
	IF stCmdModesStates.stStates.Reset THEN
		stCmdModesStates.stStates.Reset := FALSE;
		gpCh[nChanIdx]^.channel_mc_control.mode_and_state.command_w.to_mode:= HLI_IMCM_REFERENCE_MODE;
		gpCh[nChanIdx]^.channel_mc_control.mode_and_state.command_w.to_state := HLI_IMCM_PROCESS_RESETTING;		
		gpCh[nChanIdx]^.channel_mc_control.mode_and_state.command_semaphor_rw := TRUE;		
	END_IF

	HLI3_ChannelModeReference := TRUE;
ELSE
	HLI3_ChannelModeReference := FALSE;
END_IF

END_FUNCTION

// CNC/2 OperationMode/HLI3_ChannelModeStandby
FUNCTION HLI3_ChannelModeStandby : BOOL
VAR_INPUT	 
	nChanIdx: INT;
	ProgramName: STRING(HLI_IMCM_MODE_STATE_PARAM_STRL);			
END_VAR

VAR_IN_OUT
	stCmdModesStates    : ST_CNCCmdModesStates;	
END_VAR

VAR
	pString: POINTER TO STRING(HLI_IMCM_MODE_STATE_PARAM_STRL);
	nCHan: INT;
END_VAR

(* ========================================================= *)
(*    FUN: HLI_ChannelModeStandby                            *)
(* --------------------------------------------------------- *)
(*   Desc: switch channel to Standby mode / xxx              *)
(*   Author: MK, MiB, TV                                     *)
(*   Date: 16.05.2018                                        *)
(*   Rev.: 1.6                                               *)
(* ========================================================= *)

IF (NOT gpCh[nChanIdx]^.channel_mc_control.mode_and_state.command_semaphor_rw) THEN  (* only if semaphor is FALSE...... *)
	IF stCmdModesStates.stStates.Selected THEN
		stCmdModesStates.stStates.Selected := FALSE;
		gpCh[nChanIdx]^.channel_mc_control.mode_and_state.command_w.to_mode := HLI_IMCM_STANDBY_MODE;
		gpCh[nChanIdx]^.channel_mc_control.mode_and_state.command_w.to_state := HLI_IMCM_PROCESS_SELECTED;
		pString := ADR(gpCh[nChanIdx]^.channel_mc_control.mode_and_state.command_w.parameter);			
		pString^ := ProgramName;				
		gpCh[nChanIdx]^.channel_mc_control.mode_and_state.command_semaphor_rw := TRUE;		
	END_IF
	
	IF stCmdModesStates.stStates.Ready THEN
		stCmdModesStates.stStates.Ready := FALSE;
		gpCh[nChanIdx]^.channel_mc_control.mode_and_state.command_w.to_mode := HLI_IMCM_STANDBY_MODE;
		gpCh[nChanIdx]^.channel_mc_control.mode_and_state.command_w.to_state := HLI_IMCM_PROCESS_READY;		
		pString := ADR(gpCh[nChanIdx]^.channel_mc_control.mode_and_state.command_w.parameter);			
		pString^ := ProgramName;	
		gpCh[nChanIdx]^.channel_mc_control.mode_and_state.command_semaphor_rw := TRUE;		
	END_IF
	
	IF stCmdModesStates.stStates.Active THEN
		stCmdModesStates.stStates.Active := FALSE;
		gpCh[nChanIdx]^.channel_mc_control.mode_and_state.command_w.to_mode := HLI_IMCM_STANDBY_MODE;
		gpCh[nChanIdx]^.channel_mc_control.mode_and_state.command_w.to_state := HLI_IMCM_PROCESS_ACTIVE;		
		pString := ADR(gpCh[nChanIdx]^.channel_mc_control.mode_and_state.command_w.parameter);			
		pString^ := ProgramName;	
		gpCh[nChanIdx]^.channel_mc_control.mode_and_state.command_semaphor_rw := TRUE;		
	END_IF
	
	IF stCmdModesStates.stStates.Hold THEN
		stCmdModesStates.stStates.Hold := FALSE;
		gpCh[nChanIdx]^.channel_mc_control.mode_and_state.command_w.to_mode := HLI_IMCM_STANDBY_MODE;
		gpCh[nChanIdx]^.channel_mc_control.mode_and_state.command_w.to_state:= HLI_IMCM_PROCESS_HOLD;		
		gpCh[nChanIdx]^.channel_mc_control.mode_and_state.command_semaphor_rw := TRUE;	
	END_IF
	
	IF stCmdModesStates.stStates.Reset THEN
		stCmdModesStates.stStates.Reset := FALSE;
		gpCh[nChanIdx]^.channel_mc_control.mode_and_state.command_w.to_mode := HLI_IMCM_STANDBY_MODE;
		gpCh[nChanIdx]^.channel_mc_control.mode_and_state.command_w.to_state:= HLI_IMCM_PROCESS_RESETTING;		
		gpCh[nChanIdx]^.channel_mc_control.mode_and_state.command_semaphor_rw := TRUE;		
	END_IF
	
	HLI3_ChannelModeStandby := TRUE;
ELSE
	HLI3_ChannelModeStandby := FALSE;
END_IF

END_FUNCTION

// CNC/2 OperationMode/HLI3_ChannelReset
FUNCTION HLI3_ChannelReset : BOOL
VAR_INPUT
	/// Channel index 
	nChanIdx: INT;
END_VAR
VAR
	/// local pointer to Data of actual Channel 
	pChannelData: POINTER TO HIGH_LEVEL_INTERFACE_CH;
END_VAR

(* ========================================================= 	*)
(*    FUN: HLI_ChannelReset                                  	*)
(* --------------------------------------------------------- 	*)
(*   Desc:                                                   	*)
(* 	 Author: MK ,MiB, TV                                       	*)
(*   Date: 17.01.2018                                        	*)
(*   Rev.: 1.2                                               	*)
(* 	1.2 16.04.2019 Set and Reset the flag  bStateResetting in 	*)
(* 	CNCSystem structur											*)
(* ========================================================= 	*)

HLI3_ChannelReset := FALSE;
IF NOT HLI3_CheckChannelValid(nChannel := nChanIdx) THEN
	RETURN;
END_IF

(* get pointer to channel data *)
pChannelData := gpCh[nChanIdx];
IF (pChannelData = 0) THEN   (* check for zero pointer *)
	RETURN;
END_IF


CNCSystem.Channel[nChanIdx].bStateResetting := FALSE;

(* is a reset commanded *)
IF pChannelData^.bahn_lc_control.plc_reset.command_r = TRUE THEN
	
	CNCSystem.Channel[nChanIdx].bStateResetting := TRUE;

	(* Reset all M- and H-Functions whenn the channel gets resetted *)
	HLI3_ChannelResetMFunctions(nChanIdx);
	HLI3_ChannelResetHFunctions(nChanIdx);
	
	(* quit this reset *)
	pChannelData^.bahn_lc_control.plc_reset.state_w := TRUE;	
	HLI3_ChannelReset := TRUE;
END_IF

END_FUNCTION

// CNC/4 MHT-Function/HLI3_ChannelResetMFunctions
FUNCTION HLI3_ChannelResetMFunctions : BOOL
VAR_INPUT
	/// Channel number 
	nChanIdx: INT;
END_VAR
VAR
	idx: INT;
END_VAR

(* ========================================================= *)
(*    FUN: HLI_ChannelResetMFunctions                        *)
(* --------------------------------------------------------- *)
(*   Desc:                                                   *)
(* Author: MK                                                *)
(*   Date: 10.05.2007                                        *)
(*   Rev.: 1.00                                              *)
(* ========================================================= *)

IF NOT HLI3_CheckChannelValid(nChannel := nChanIdx) THEN
	HLI3_ChannelResetMFunctions := FALSE;
	RETURN; (* A b b r u c h *)
END_IF


FOR idx := 1 TO 999 DO
	CNCSystem.Channel[nChanIdx].M[idx].bState_rw := FALSE;
	CNCSystem.Channel[nChanIdx].M[idx].bRes := FALSE;
	CNCSystem.Channel[nChanIdx].actM_r :='';
END_FOR

HLI3_ChannelResetMFunctions := TRUE;

END_FUNCTION

// CNC/4 MHT-Function/HLI3_ChannelResetHFunctions
FUNCTION HLI3_ChannelResetHFunctions : BOOL
VAR_INPUT
	/// Channel number 
	nChanIdx: INT;
END_VAR
VAR
	idx: INT;
END_VAR

(* ========================================================= *)
(*    FUN: HLI_ChannelResetHFunctions                        *)
(* --------------------------------------------------------- *)
(*   Desc:                                                   *)
(* Author: MiB                                                *)
(*   Date: 23.11.2012                                        *)
(*   Rev.: 1.1                                              *)
(* ========================================================= *)



IF NOT HLI3_CheckChannelValid(nChannel := nChanIdx) THEN
	HLI3_ChannelResetHFunctions := FALSE;
	RETURN; (* A b b r u c h *)
END_IF


FOR idx := 0 TO 999 DO
	CNCSystem.Channel[nChanIdx].H[idx].bState_rw := FALSE;
	CNCSystem.Channel[nChanIdx].H[idx].bRes := FALSE;
	CNCSystem.Channel[nChanIdx].actH_r :='';
END_FOR

HLI3_ChannelResetHFunctions := TRUE;

END_FUNCTION

// CNC/2 OperationMode/HLI3_ChannelResetRequest
FUNCTION_BLOCK HLI3_ChannelResetRequest
VAR_INPUT
	bExec: BOOL;
	/// Channel number 
	nChanIdx: INT;
	pChannel: POINTER TO ST_CncChannel;
END_VAR
VAR_OUTPUT
	bBusy: BOOL;
	bSwitchMode: BOOL;
	nMode: UDINT;
END_VAR
VAR
	fbRtrigExec: R_TRIG;
	/// Index of channel specific HLI area 
	nHliChIfcIdx: INT;
	nState: UINT;
	pCommand: POINTER TO HLI_PROC_TRANS_TO_MODE_STATE;
	actualMode: UDINT;
	fbTON: TON;
END_VAR

(******************************************************************************)
(* POU:				HLI_ChannelResetRequest									*)
(* Type:				Function block										*)
(* Customer:		Common													*)
(* Date:				07/11/16											*)
(* Last:				10/03/10											*)
(* -------------------------------------------------------------------------- *)
(* Revision:		1.0														*)
(* Author:			MiB														*)
(* Description: 	Performs a reset in the given cnc channel. 				*)
(* -------------------------------------------------------------------------- *)
(* Revision:		1.10													*)
(* Author:			MiB														*)
(* Description: 	Changed from PRG to FB.									*)
(* -------------------------------------------------------------------------- *)
(* Revision:		2.00															*)
(* Author:			HR																*)
(* Description: 	Deleted references to global variable 'PLCMachineMode[n]'.		*)
(*						The FB now works with VAR_OUTPUT 'nMode' and 'bSwitchMode'	*)
(*						as a callback to the initiator to let it perform the change	*)
(*						of the operation mode by itself in order to reset the cnc	*)
(*						channel.													*)
(* -------------------------------------------------------------------------- *)
(* Revision:		2.01																			*)
(* Author:			TV																				*)
(* Description: 	Expand State "Wait for previous mode"  *)
(*				Prevent to trigger the state machine during the mode switch							*)
(* -------------------------------------------------------------------------- *)
(* Revision:		2.02																			*)
(* Author:			MiB																				*)
(* Description: 	Tc3*)
(******************************************************************************)


fbRtrigExec( clk := bExec   );

IF fbRtrigExec.Q THEN
	bBusy := TRUE;
	nState := 10;
END_IF


CASE nState OF

0:		(* IDLE *)
		bBusy := FALSE;

10:	(* Reset request: get actual opmode *)
		bSwitchMode := FALSE;
		actualMode := gpCh[nChanIdx]^.channel_mc_control.mode_and_state.state_r.mode;
		nState := nState + 10;

20:  (* switch to standby *)
		bSwitchMode := TRUE;
		nMode:= HLI_IMCM_STANDBY_MODE;
		fbTON(IN:= FALSE);
		nState := nState + 10;

30: 	(* Wait for modeswitch *)
		bSwitchMode := FALSE;
		fbTON(IN:= TRUE, PT:= t#2000ms);
	 	IF gpCh[nChanIdx]^.channel_mc_control.mode_and_state.state_r.mode = HLI_IMCM_STANDBY_MODE THEN
			nState := nState + 10;
		END_IF
		IF fbTON.Q THEN
			(* Timeout Error -> go on with next step *)
			nState := nState + 10;
		END_IF

40:	(* switch back to previous mode *)
		bSwitchMode := TRUE;
		nMode:= actualMode;
		fbTON(IN:= FALSE);
		nState := nState + 10;

50:	(* Wait for previous mode  *)
		fbTON(IN:= TRUE, PT:= t#2000ms);
		IF (gpCh[nChanIdx]^.channel_mc_control.mode_and_state.state_r.mode = 	actualMode) THEN
			nState := nState + 10;
		END_IF
		IF fbTON.Q THEN
			(* Timeout Error -> go on with next step *)
			nState := nState + 10;
		END_IF

60: 	(* ready *)
		bSwitchMode := FALSE;
		nState := 0;

END_CASE



(* das muss ins aufrufende Programm: (HLI_CNCChannel)

VAR
	bResetRequest:			BOOL;
	fbRTrigReset:			R_TRIG;
	ChannelResetRequest: HLI_ChannelResetRequest;
END_VAR

fbRTrigReset(clk := bStateReset);
IF fbRTrigReset.Q THEN
	bResetRequest := TRUE;
	...
END_IF

(* Handle Channel reset *)
ChannelResetRequest
	(bExec 		:= bResetRequest ,
	 nChan 		:= nChan,
	 pChannel	:= ADR(CNCSystem.Channel[nChan])
	);

IF ChannelResetRequest.bSwitchMode THEN
	bModeStandby	:= bModeStandby OR (ChannelResetRequest.nMode = HLI_IMCM_STANDBY_MODE);
	bModeAutomatic	:= bModeAutomatic OR (ChannelResetRequest.nMode = HLI_IMCM_AUTOMATIC_MODE);
	bModeManual		:= bModeManual OR (ChannelResetRequest.nMode = HLI_IMCM_MANUAL_MODE);
	bModeMDI			:= bModeMDI OR (ChannelResetRequest.nMode = HLI_IMCM_MDI_MODE);
	bModeReference	:= bModeReference OR (ChannelResetRequest.nMode = HLI_IMCM_REFERENCE_MODE);
END_IF

IF bResetRequest AND NOT ChannelResetRequest.bBusy THEN
	bResetRequest := FALSE;
END_IF

*)

END_FUNCTION_BLOCK

// CNC/2 OperationMode/HLI3_CNCChannel
FUNCTION_BLOCK HLI3_CNCChannel
VAR_INPUT
	/// index of channel
	nChanIdx: INT;
 
	bCmdAutomatic : BOOL;
	bCmdManual : BOOL;
    bCmdReference : BOOL;
    bCmdMDI : BOOL;		
	bCmdStandby: BOOL;
	bCmdStart : BOOL;
	bCmdStop  : BOOL;
	bCmdReset : BOOL;		
	/// must be xxx.nc 
	sProgramName: STRING(HLI_IMCM_MODE_STATE_PARAM_STRL);
	/// the MDI string 
	sMDIString: STRING(HLI_IMCM_MODE_STATE_PARAM_STRL);
	/// static signal 
	bBackwardMotion: BOOL;
	/// static signal 
	bFeedHold: BOOL;
	/// static signal 
	bReducedFeed: BOOL;
	/// static signal 
	bSingleBlock: BOOL;
	/// static signal 
	bPrgBlockIgnore: BOOL;
	/// static signal 
	bM01Stop: BOOL;
	/// static signal 
	nSyntaxCheck: DINT;		
	// Manual Mode
	stManualModeParameter: ST_ManualModeParameter;
	stManualModeControlElements: ST_ManualModeControlElements;
	// M30 Acknowledgement inside Channel FB
	bM30Acknowledgement : BOOL;
	// Override 
	nFeedOverride : UINT;
	nRapidFeedOverride : UINT;
	bEmergencyStop : BOOL;
	stOptions : ST_CNC_CH_Options;
END_VAR
VAR_IN_OUT
	/// please only a flank 
	bModeStandby: BOOL;
	/// please only a flank 
	bModeAutomatic: BOOL;
	/// please only a flank 
	bModeManual: BOOL;
	/// please only a flank 
	bModeMDI: BOOL;
	/// please only a flank 
	bModeReference: BOOL;
	/// please only a flank 
	bStateSelect: BOOL;
	/// please only a flank 
	bStateReady: BOOL;
	/// please only a flank 
	bStateStart: BOOL;
	/// please only a flank 
	bStateStop: BOOL;
	/// please only a flank 
	bStateReset: BOOL;
	/// please only a flank 
	bDoSingleBlock: BOOL;
	// manual mode
	stManualModeControlElementState: ST_ManualModeControlElementState;
END_VAR
VAR
	bGoToActive	: BOOL;	 	
	/// Pointer to channel control structure 
	pChannel: POINTER TO ST_CncChannel;
	ChannelMHTFunction: HLI3_QuitChannelMHTFunction;
	/// Current Mode of Operation Modes;
	currentMode: UDINT;
	/// Current State of Operation Modes;
	currentState: UDINT;
	idx: INT;	
	bCheckOpModeFirst: BOOL;
	fbRTrigReset: R_TRIG;
	bResetRequest: BOOL;	
	nStateAutoMDIStart: INT;
	ModeManual : HLI3_ManualModeHandler;	
	stCmdModesStates    : ST_CNCCmdModesStates;

	fbRTrigCmdStart: R_TRIG;
	fbRTrigCmdStop:  R_TRIG;
	fbRTrigCmdReset: R_TRIG;	
	fbRTrigCmdAutomatic : R_TRIG;
	fbRTrigCmdManual : R_TRIG;
    fbRTrigCmdReference : R_TRIG;
    fbRTrigCmdMDI : R_TRIG;		
	fbRTrigCmdStandby: R_TRIG;
END_VAR

